// TIA Portal V20 export
FUNCTION_BLOCK "CallEquipment"   // FB8, LAD
TITLE = CallEquipment
AUTHOR : ERsystem_FA2_DH. Kim
// This block contains the logic and futher calls (e.g. sequences, control modules, diagnostics etc.) of the equipment module.
// stored: IsIECCheckEnabled true, MemoryReserve 100, Namespace Unit1.Em0, SetENOAutomatically false
   VAR_INPUT
      ZoneOperationEnable { ExternalWritable := 'False'} : "LWONIK_typeSafetyZoneManualOperation";
   END_VAR
   VAR_IN_OUT
      unitStatus : "LAF_typeUnitStatus";   // Current unit status o be used in this EM
      unitAlarmDB : "LAF_typeAlarms";   // Summarized EM Alarms for the Unit
      emFeedback : "LUC_typeEmFeedback";   // Feedback of the EM to the Unit
   END_VAR
   VAR
      instSequenceUnwinder { S7_SetPoint := 'True'} : "Unit1.Em0.Sequence_1_SepaUnwinderTop";
      instTopHomeJob1 { S7_SetPoint := 'True'} : "LAF_SelectJob";
      instTopUnwindingJob2 { S7_SetPoint := 'True'} : "LAF_SelectJob";
      instTopStopJob3 { S7_SetPoint := 'True'} : "LAF_SelectJob";
      instTopRewidnigJob4 { S7_SetPoint := 'True'} : "LAF_SelectJob";
      instTopRewidnigJob10 { S7_SetPoint := 'True'} : "LAF_SelectJob";
      instCmTopDirectionCheckSensor { S7_SetPoint := 'True'} : "LBC_DigitalSignalCn";
      instCmUnwinderTopRadiusMeasure { ExternalAccessible := 'False'; ExternalVisible := 'False'; ExternalWritable := 'False'} : "LBC_AnalogInputCn";
      instCmRadiusMeasure { S7_SetPoint := 'True'} : "LER_RadiusMeasure";
      instCmUnwinderTopAxisB { S7_SetPoint := 'True'} : "LBC_Axis64Pos_TecPlcCn";
      instInterlockCmUnwinderTopAxisB { S7_SetPoint := 'True'} : "LER_Axis64Pos_InterlockSummary";
      instCmUnwinderAirShaftTopOnOff { ExternalAccessible := 'False'; ExternalVisible := 'False'; ExternalWritable := 'False'; S7_SetPoint := 'True'} : "LBC_TwoWayActuatorCn";
      instCmUnwinderTopEpcControllerInterface { ExternalAccessible := 'False'; ExternalVisible := 'False'; ExternalWritable := 'False'; S7_SetPoint := 'True'} : "LER_EPC_CON600";
      instManageAlarms { ExternalWritable := 'False'} : "LAF_ManageAlarms";
      instEventsPFE : "Unit1.Em0.EventsPFE";
      instLER_BrakeTestUnwinderTopAxisB { S7_SetPoint := 'True'} : "LER_BrakeTest";
      statUnitStatus { ExternalWritable := 'False'} : "LAF_typeUnitStatus";   // Unit Status used in this EM
      statSlmStatus : Struct
         running { ExternalWritable := 'False'} : Bool;
         powerOff { ExternalWritable := 'False'} : Bool;
      END_STRUCT;
      statAllBrakeTest { ExternalWritable := 'False'} : "LER_typeBrakeTestUnitCommands";
      statTonTime { ExternalAccessible := 'False'; ExternalVisible := 'False'; ExternalWritable := 'False'} : Array[0..1999] of TON_TIME;
      statTofTime { ExternalAccessible := 'False'; ExternalVisible := 'False'; ExternalWritable := 'False'} : Array[0..99] of TOF_TIME;
      statPulse { ExternalAccessible := 'False'; ExternalVisible := 'False'; ExternalWritable := 'False'} : Struct
         miscellaneous : Array[0..99] of Bool;
         workingDone : Struct
            mainPnP : Array[0..99] of Bool;
            alignTable : Array[0..99] of Bool;
            ngPnP : Array[0..99] of Bool;
         END_STRUCT;
         axisEnable : Array[0..99] of Bool;
         brakeTest : Array[0..99] of Bool;
      END_STRUCT;
      statEnableManualCmds : Bool;
      statRcEnableCmds : Bool;
      Scan_on { ExternalAccessible := 'False'; ExternalVisible := 'False'; ExternalWritable := 'False'} : Bool;
      "*** Interlock Axis ***" { ExternalAccessible := 'False'; ExternalVisible := 'False'; ExternalWritable := 'False'} : Bool;
      "UnwinderTopAxisB Home" { S7_SetPoint := 'True'} : "Homing.LER_Axis";
      "UnwinderTopAxisB Jog_CW" { S7_SetPoint := 'True'} : "Jog.LER_Axis";
      "UnwinderTopAxisB Jog_CCW" { S7_SetPoint := 'True'} : "Jog.LER_Axis";
      "UnwinderTopAxisB Position" { S7_SetPoint := 'True'} : Array[0..5] of "Position.LER_Axis";
      "*** Interlock Actuator ******" { ExternalAccessible := 'False'; ExternalVisible := 'False'; ExternalWritable := 'False'} : Bool;
      "UnwinderAirShaftTop On" { S7_SetPoint := 'True'} : "Cylinder.LER_Actuator";
      "UnwinderAirShaftTop Off" { S7_SetPoint := 'True'} : "Cylinder.LER_Actuator";
      AXIS1 : "LER_CM_Name";
      Cylinder1 : "LER_CM_Name";
      citi_Ptrig : Array[0..20] of Bool;
      citiTon : Array[0..20] of TON_TIME;
      citi : Time;
      citiTest : Array[0..20] of Bool;
   END_VAR
   VAR_TEMP
      tempIndex : Int;
      tempScInProduction : Bool;   // Mode Production and StateComplete
      tempScNoProduction : Bool;   // Mode Manual and StateComplete
   END_VAR
   VAR CONSTANT
      delayTime : Time := T#3s;
      TRUE : Bool := TRUE;
      FALSE : Bool := FALSE;
      NO_JOB : DInt;   // No job
      MIN_POSITION_NUMBER : SInt;
      INIT_POSITION_NUMBER : SInt := -1;
   END_VAR
   VAR_TEMP   // added for the SCL form of the ladder/FBD networks
      _w1 : Bool;
      _w2 : Bool;
      _w3 : Bool;
      _w4 : Bool;
      _w5 : Bool;
      _w6 : Bool;
      _w7 : Bool;
      _w8 : Bool;
      _w9 : Bool;
   END_VAR
BEGIN

REGION Network 1: BLOCK INFO HEADER
   // (company) / (C) Copyright (year)
   // ---------------------------------------------------------------------------------
   // Title:                             (Title of this block)
   // Comment/Function: (that is implemented in the block)
   // Library/Family:           (that the source is dedicated to)
   // Author:                        (department / person in charge / contact)
   // Target System:          (test system with FW version)
   // Engineering:              TIA Portal (SW version)
   // Restrictions:               (OB types, etc.)
   // Requirements:           (hardware, technological package, etc.)
   // ---------------------------------------------------------------------------------
   // Change log table:
   // Version          | Date             | Signature      | Expert in charge  | Changes applied ------------------------|----------------------|-------------------------|--------------------------------|-----------------------
   // 001.000.000 | yyyy-mm-dd | 0x00000000 | (name of expert) | First released version
END_REGION

REGION Network 2: DESCRIPTION
   // This is a template block provided by the Automation Framework. It can be used to create an own project.
   // The Block Info Header is prepared to put in your own data.
   // Description of the block could be added here and the docu created by Code2Docu.
END_REGION

REGION Network 3: disableFeedbackHomePos
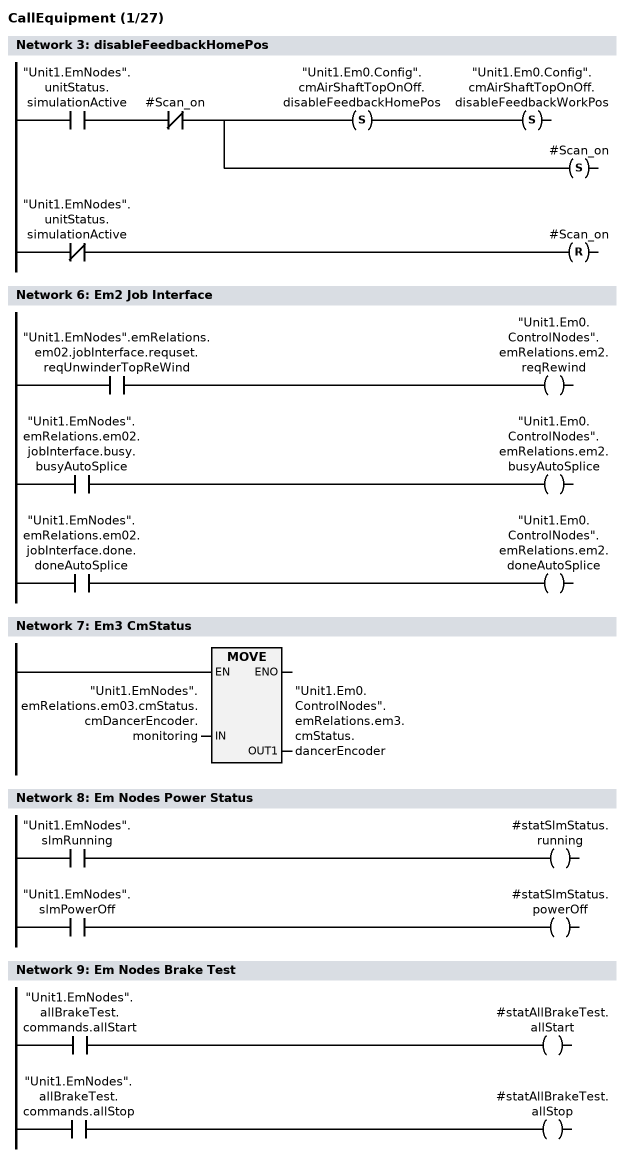
   RUNG wire#powerrail
      Contact( "Unit1.EmNodes".unitStatus.simulationActive )
      I_Contact( #Scan_on )
      wire#w1
      S_Coil( "Unit1.Em0.Config".cmAirShaftTopOnOff.disableFeedbackHomePos )
      S_Coil( "Unit1.Em0.Config".cmAirShaftTopOnOff.disableFeedbackWorkPos )
   END_RUNG
   RUNG wire#w1
      S_Coil( #Scan_on )
   END_RUNG
   RUNG wire#powerrail
      I_Contact( "Unit1.EmNodes".unitStatus.simulationActive )
      R_Coil( #Scan_on )
   END_RUNG
   // the same network as SCL:
   IF "Unit1.EmNodes".unitStatus.simulationActive AND NOT #Scan_on THEN
       "Unit1.Em0.Config".cmAirShaftTopOnOff.disableFeedbackHomePos := TRUE;
       "Unit1.Em0.Config".cmAirShaftTopOnOff.disableFeedbackWorkPos := TRUE;
       #Scan_on := TRUE;
   END_IF;
   IF NOT "Unit1.EmNodes".unitStatus.simulationActive THEN #Scan_on := FALSE; END_IF;
END_REGION

REGION Network 4: ******************** Unit Input ********************
END_REGION

REGION Network 5: Em2 Sequence Interface
END_REGION

REGION Network 6: Em2 Job Interface
   RUNG wire#powerrail
      Contact( "Unit1.EmNodes".emRelations.em02.jobInterface.requset.reqUnwinderTopReWind )
      Coil( "Unit1.Em0.ControlNodes".emRelations.em2.reqRewind )
   END_RUNG
   RUNG wire#powerrail
      Contact( "Unit1.EmNodes".emRelations.em02.jobInterface.busy.busyAutoSplice )
      Coil( "Unit1.Em0.ControlNodes".emRelations.em2.busyAutoSplice )
   END_RUNG
   RUNG wire#powerrail
      Contact( "Unit1.EmNodes".emRelations.em02.jobInterface.done.doneAutoSplice )
      Coil( "Unit1.Em0.ControlNodes".emRelations.em2.doneAutoSplice )
   END_RUNG
   // the same network as SCL:
   "Unit1.Em0.ControlNodes".emRelations.em2.reqRewind := "Unit1.EmNodes".emRelations.em02.jobInterface.requset.reqUnwinderTopReWind;
   "Unit1.Em0.ControlNodes".emRelations.em2.busyAutoSplice := "Unit1.EmNodes".emRelations.em02.jobInterface.busy.busyAutoSplice;
   "Unit1.Em0.ControlNodes".emRelations.em2.doneAutoSplice := "Unit1.EmNodes".emRelations.em02.jobInterface.done.doneAutoSplice;
END_REGION

REGION Network 7: Em3 CmStatus
   RUNG wire#powerrail
      Move(in := "Unit1.EmNodes".emRelations.em03.cmStatus.cmDancerEncoder.monitoring, out1 => "Unit1.Em0.ControlNodes".emRelations.em3.cmStatus.dancerEncoder)
   END_RUNG
   // the same network as SCL:
   "Unit1.Em0.ControlNodes".emRelations.em3.cmStatus.dancerEncoder := "Unit1.EmNodes".emRelations.em03.cmStatus.cmDancerEncoder.monitoring;
END_REGION

REGION Network 8: Em Nodes Power Status
   RUNG wire#powerrail
      Contact( "Unit1.EmNodes".slmRunning )
      Coil( #statSlmStatus.running )
   END_RUNG
   RUNG wire#powerrail
      Contact( "Unit1.EmNodes".slmPowerOff )
      Coil( #statSlmStatus.powerOff )
   END_RUNG
   // the same network as SCL:
   #statSlmStatus.running := "Unit1.EmNodes".slmRunning;
   #statSlmStatus.powerOff := "Unit1.EmNodes".slmPowerOff;
END_REGION

REGION Network 9: Em Nodes Brake Test
   RUNG wire#powerrail
      Contact( "Unit1.EmNodes".allBrakeTest.commands.allStart )
      Coil( #statAllBrakeTest.allStart )
   END_RUNG
   RUNG wire#powerrail
      Contact( "Unit1.EmNodes".allBrakeTest.commands.allStop )
      Coil( #statAllBrakeTest.allStop )
   END_RUNG
   // the same network as SCL:
   #statAllBrakeTest.allStart := "Unit1.EmNodes".allBrakeTest.commands.allStart;
   #statAllBrakeTest.allStop := "Unit1.EmNodes".allBrakeTest.commands.allStop;
END_REGION

REGION Network 10: *************** Equipment Control **************************
END_REGION

REGION Network 11: Interlink EM to Unit
   // This block links and unlinks the EM from the unit. The command to link/unlink can be set directly by the inputs of the block (e.g. to link/unlink based on any program logic) or through the InOut "hmiInterface". The block changes the output "isLinked" to true/false, depending on the command and if a change is allowed. A changed is allowed if the unit is in state aborted, clearing or stopped. The output "isLinked" is send back to the unit. If the EM is not linked, the unit ignores this EM.
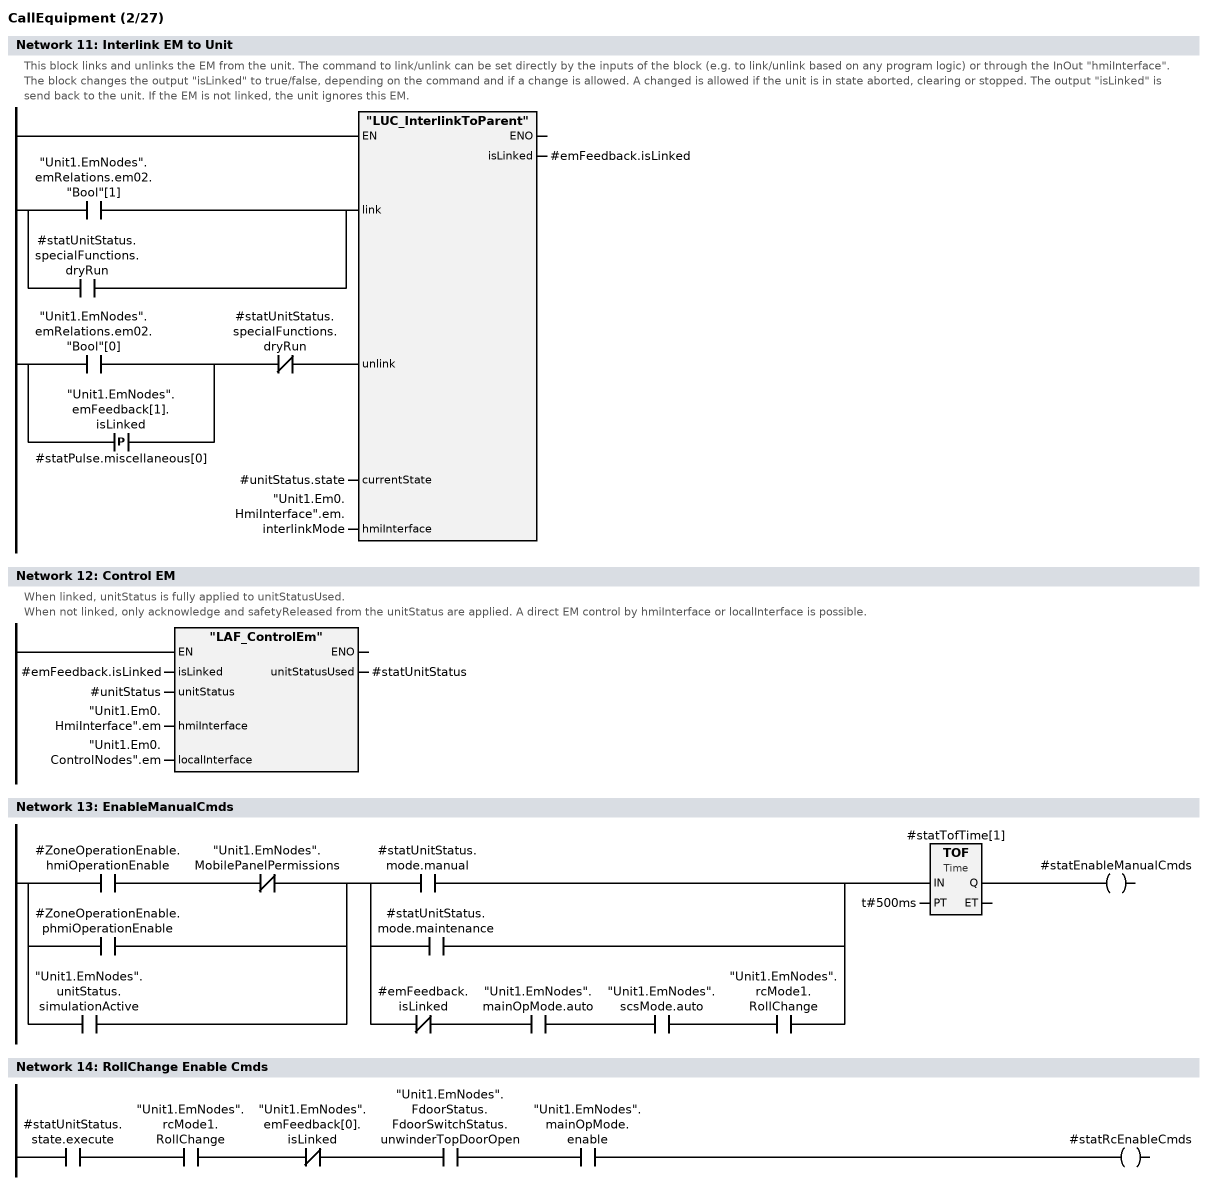
   RUNG wire#powerrail
      "LUC_InterlinkToParent"(link := wire#w1, unlink := wire#w3, currentState := #unitStatus.state, hmiInterface := "Unit1.Em0.HmiInterface".em.interlinkMode, isLinked => #emFeedback.isLinked)
   END_RUNG
   RUNG wire#powerrail
      Contact( "Unit1.EmNodes".emRelations.em02."Bool"[1] )
   END_RUNG wire#w1
   RUNG wire#powerrail
      Contact( #statUnitStatus.specialFunctions.dryRun )
   END_RUNG wire#w1
   RUNG wire#powerrail
      Contact( "Unit1.EmNodes".emRelations.em02."Bool"[0] )
      wire#w2
      I_Contact( #statUnitStatus.specialFunctions.dryRun )
   END_RUNG wire#w3
   RUNG wire#powerrail
      P_Contact(operand := "Unit1.EmNodes".emFeedback[1].isLinked, bit := #statPulse.miscellaneous[0])
   END_RUNG wire#w2
   // the same network as SCL:
   #_w1 := "Unit1.EmNodes".emFeedback[1].isLinked AND NOT #statPulse.miscellaneous[0];   // rising edge of "Unit1.EmNodes".emFeedback[1].isLinked
   #statPulse.miscellaneous[0] := "Unit1.EmNodes".emFeedback[1].isLinked;
   "LUC_InterlinkToParent"(link := "Unit1.EmNodes".emRelations.em02."Bool"[1] OR #statUnitStatus.specialFunctions.dryRun,
                           unlink := ("Unit1.EmNodes".emRelations.em02."Bool"[0] OR #_w1) AND NOT #statUnitStatus.specialFunctions.dryRun,
                           currentState := #unitStatus.state,
                           hmiInterface := "Unit1.Em0.HmiInterface".em.interlinkMode,
                           isLinked => #emFeedback.isLinked);
END_REGION

REGION Network 12: Control EM
   // When linked, unitStatus is fully applied to unitStatusUsed.
   // When not linked, only acknowledge and safetyReleased from the unitStatus are applied. A direct EM control by hmiInterface or localInterface is possible.
   RUNG wire#powerrail
      "LAF_ControlEm"(isLinked := #emFeedback.isLinked, unitStatus := #unitStatus, hmiInterface := "Unit1.Em0.HmiInterface".em, localInterface := "Unit1.Em0.ControlNodes".em, unitStatusUsed => #statUnitStatus)
   END_RUNG
   // the same network as SCL:
   "LAF_ControlEm"(isLinked := #emFeedback.isLinked,
                   unitStatus := #unitStatus,
                   hmiInterface := "Unit1.Em0.HmiInterface".em,
                   localInterface := "Unit1.Em0.ControlNodes".em,
                   unitStatusUsed => #statUnitStatus);
END_REGION

REGION Network 13: EnableManualCmds
   RUNG wire#powerrail
      Contact( #ZoneOperationEnable.hmiOperationEnable )
      I_Contact( "Unit1.EmNodes".MobilePanelPermissions )
      wire#w1
      Contact( #statUnitStatus.mode.manual )
      wire#w2
      { S7_Templates := "time_type := Time" } #statTofTime[1].TOF(pt := t#500ms, et =>)
      Coil( #statEnableManualCmds )
   END_RUNG
   RUNG wire#powerrail
      Contact( #ZoneOperationEnable.phmiOperationEnable )
   END_RUNG wire#w1
   RUNG wire#powerrail
      Contact( "Unit1.EmNodes".unitStatus.simulationActive )
   END_RUNG wire#w1
   RUNG wire#w1
      Contact( #statUnitStatus.mode.maintenance )
   END_RUNG wire#w2
   RUNG wire#w1
      I_Contact( #emFeedback.isLinked )
      Contact( "Unit1.EmNodes".mainOpMode.auto )
      Contact( "Unit1.EmNodes".scsMode.auto )
      Contact( "Unit1.EmNodes".rcMode1.RollChange )
   END_RUNG wire#w2
   // the same network as SCL:
   #statTofTime[1].TOF(IN := ((#ZoneOperationEnable.hmiOperationEnable AND NOT "Unit1.EmNodes".MobilePanelPermissions) OR #ZoneOperationEnable.phmiOperationEnable OR "Unit1.EmNodes".unitStatus.simulationActive) AND (#statUnitStatus.mode.manual OR #statUnitStatus.mode.maintenance OR (NOT #emFeedback.isLinked AND "Unit1.EmNodes".mainOpMode.auto AND "Unit1.EmNodes".scsMode.auto AND "Unit1.EmNodes".rcMode1.RollChange)),
                       PT := t#500ms);
   #statEnableManualCmds := #statTofTime[1].Q;
END_REGION

REGION Network 14: RollChange Enable Cmds
   RUNG wire#powerrail
      Contact( #statUnitStatus.state.execute )
      Contact( "Unit1.EmNodes".rcMode1.RollChange )
      I_Contact( "Unit1.EmNodes".emFeedback[0].isLinked )
      Contact( "Unit1.EmNodes".FdoorStatus.FdoorSwitchStatus.unwinderTopDoorOpen )
      Contact( "Unit1.EmNodes".mainOpMode.enable )
      Coil( #statRcEnableCmds )
   END_RUNG
   // the same network as SCL:
   #statRcEnableCmds := #statUnitStatus.state.execute AND "Unit1.EmNodes".rcMode1.RollChange AND NOT "Unit1.EmNodes".emFeedback[0].isLinked AND "Unit1.EmNodes".FdoorStatus.FdoorSwitchStatus.unwinderTopDoorOpen AND "Unit1.EmNodes".mainOpMode.enable;
END_REGION

REGION Network 15: *************** Control Modules (Sensors) ********************
   // Call control modules that are sensors before the em logic (jobs and sequence), so that the latest value is used in the logic.
END_REGION

REGION Network 16: Call instCmTopDirectionCheckSensor (LBC_DigitalSignal)
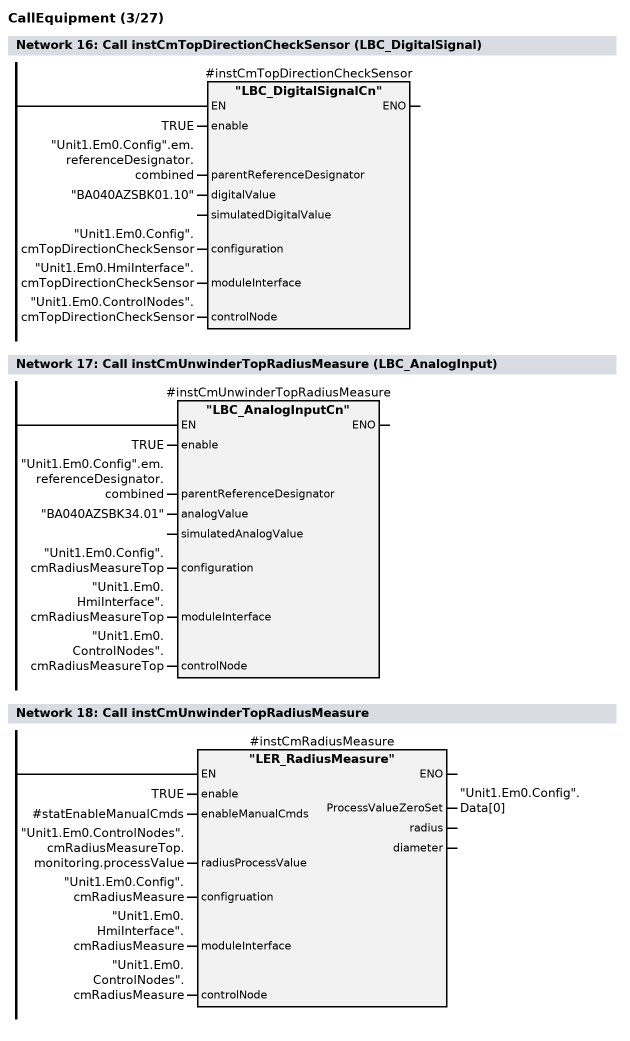
   RUNG wire#powerrail
      #instCmTopDirectionCheckSensor(enable := TRUE, parentReferenceDesignator := "Unit1.Em0.Config".em.referenceDesignator.combined, digitalValue := "BA040AZSBK01.10", simulatedDigitalValue :=, configuration := "Unit1.Em0.Config".cmTopDirectionCheckSensor, moduleInterface := "Unit1.Em0.HmiInterface".cmTopDirectionCheckSensor, controlNode := "Unit1.Em0.ControlNodes".cmTopDirectionCheckSensor)
   END_RUNG
   // the same network as SCL:
   #instCmTopDirectionCheckSensor(enable := TRUE,   // "LBC_DigitalSignalCn"
                           parentReferenceDesignator := "Unit1.Em0.Config".em.referenceDesignator.combined,
                           digitalValue := "BA040AZSBK01.10",
                           configuration := "Unit1.Em0.Config".cmTopDirectionCheckSensor,
                           moduleInterface := "Unit1.Em0.HmiInterface".cmTopDirectionCheckSensor,
                           controlNode := "Unit1.Em0.ControlNodes".cmTopDirectionCheckSensor);
END_REGION

REGION Network 17: Call instCmUnwinderTopRadiusMeasure (LBC_AnalogInput)
   RUNG wire#powerrail
      #instCmUnwinderTopRadiusMeasure(enable := TRUE, parentReferenceDesignator := "Unit1.Em0.Config".em.referenceDesignator.combined, analogValue := "BA040AZSBK34.01", simulatedAnalogValue :=, configuration := "Unit1.Em0.Config".cmRadiusMeasureTop, moduleInterface := "Unit1.Em0.HmiInterface".cmRadiusMeasureTop, controlNode := "Unit1.Em0.ControlNodes".cmRadiusMeasureTop)
   END_RUNG
   // the same network as SCL:
   #instCmUnwinderTopRadiusMeasure(enable := TRUE,   // "LBC_AnalogInputCn"
                           parentReferenceDesignator := "Unit1.Em0.Config".em.referenceDesignator.combined,
                           analogValue := "BA040AZSBK34.01",
                           configuration := "Unit1.Em0.Config".cmRadiusMeasureTop,
                           moduleInterface := "Unit1.Em0.HmiInterface".cmRadiusMeasureTop,
                           controlNode := "Unit1.Em0.ControlNodes".cmRadiusMeasureTop);
END_REGION

REGION Network 18: Call instCmUnwinderTopRadiusMeasure
   RUNG wire#powerrail
      #instCmRadiusMeasure(enable := TRUE, enableManualCmds := #statEnableManualCmds, radiusProcessValue := "Unit1.Em0.ControlNodes".cmRadiusMeasureTop.monitoring.processValue, configruation := "Unit1.Em0.Config".cmRadiusMeasure, moduleInterface := "Unit1.Em0.HmiInterface".cmRadiusMeasure, controlNode := "Unit1.Em0.ControlNodes".cmRadiusMeasure, ProcessValueZeroSet => "Unit1.Em0.Config".Data[0], radius =>, diameter =>)
   END_RUNG
   // the same network as SCL:
   #instCmRadiusMeasure(enable := TRUE,   // "LER_RadiusMeasure"
                        enableManualCmds := #statEnableManualCmds,
                        radiusProcessValue := "Unit1.Em0.ControlNodes".cmRadiusMeasureTop.monitoring.processValue,
                        configruation := "Unit1.Em0.Config".cmRadiusMeasure,
                        moduleInterface := "Unit1.Em0.HmiInterface".cmRadiusMeasure,
                        controlNode := "Unit1.Em0.ControlNodes".cmRadiusMeasure,
                        ProcessValueZeroSet => "Unit1.Em0.Config".Data[0]);
END_REGION

REGION Network 19: *************** Equipment Logic ***************************
END_REGION

REGION Network 20: Map Unit Status to Sequence Status
   // This block maps the unit status to the seuqnce status. Thus, it controls the sequence depending on the unit status. E.g. it sets the sequence to automatic when the unit state is in productions. This blocks work perfectly with the sequences provided in the AF. 
   // This typed block (MapUnitStatusToSequence) could be adjusted to specific application requirements or if other, user-defined sequences are used.
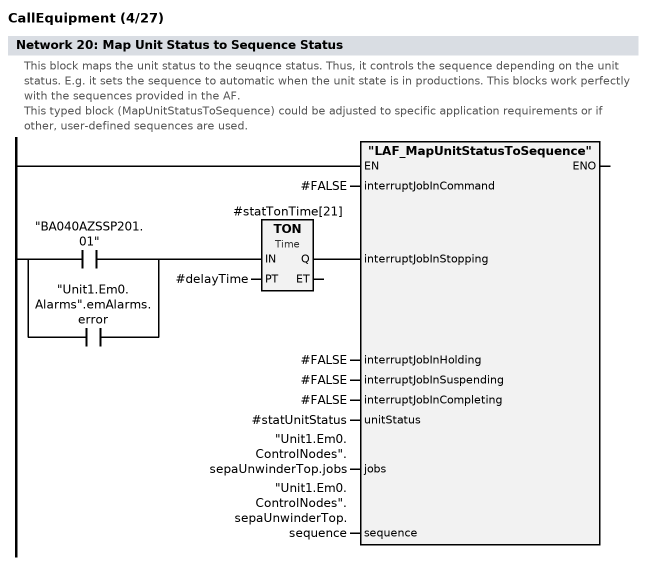
   RUNG wire#powerrail
      "LAF_MapUnitStatusToSequence"(interruptJobInStopping := wire#w2, interruptJobInCommand := #FALSE, interruptJobInHolding := #FALSE, interruptJobInSuspending := #FALSE, interruptJobInCompleting := #FALSE, unitStatus := #statUnitStatus, jobs := "Unit1.Em0.ControlNodes".sepaUnwinderTop.jobs, sequence := "Unit1.Em0.ControlNodes".sepaUnwinderTop.sequence)
   END_RUNG
   RUNG wire#powerrail
      Contact( "BA040AZSSP201.01" )
      wire#w1
      { S7_Templates := "time_type := Time" } #statTonTime[21].TON(pt := #delayTime, et =>)
   END_RUNG wire#w2
   RUNG wire#powerrail
      Contact( "Unit1.Em0.Alarms".emAlarms.error )
   END_RUNG wire#w1
   // the same network as SCL:
   #statTonTime[21].TON(IN := "BA040AZSSP201.01" OR "Unit1.Em0.Alarms".emAlarms.error, PT := #delayTime);
   "LAF_MapUnitStatusToSequence"(interruptJobInCommand := #FALSE,
                           interruptJobInStopping := #statTonTime[21].Q,
                           interruptJobInHolding := #FALSE,
                           interruptJobInSuspending := #FALSE,
                           interruptJobInCompleting := #FALSE,
                           unitStatus := #statUnitStatus,
                           jobs := "Unit1.Em0.ControlNodes".sepaUnwinderTop.jobs,
                           sequence := "Unit1.Em0.ControlNodes".sepaUnwinderTop.sequence);
END_REGION

REGION Network 22: Unwinder Top Select Job
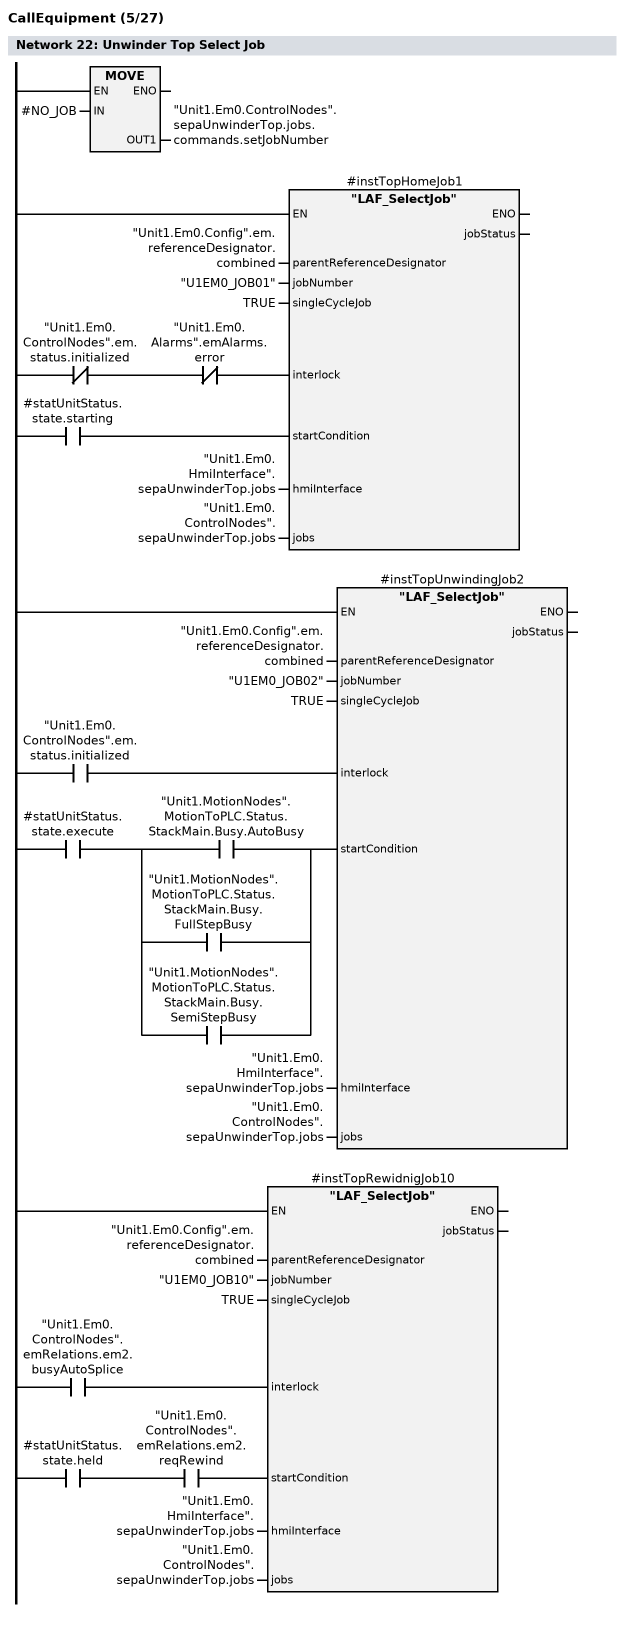
   RUNG wire#powerrail
      Move(in := #NO_JOB, out1 => "Unit1.Em0.ControlNodes".sepaUnwinderTop.jobs.commands.setJobNumber)
   END_RUNG
   RUNG wire#powerrail
      #instTopHomeJob1(interlock := wire#w1, startCondition := wire#w2, parentReferenceDesignator := "Unit1.Em0.Config".em.referenceDesignator.combined, jobNumber := "U1EM0_JOB01", singleCycleJob := TRUE, hmiInterface := "Unit1.Em0.HmiInterface".sepaUnwinderTop.jobs, jobs := "Unit1.Em0.ControlNodes".sepaUnwinderTop.jobs, jobStatus =>)
   END_RUNG
   RUNG wire#powerrail
      I_Contact( "Unit1.Em0.ControlNodes".em.status.initialized )
      I_Contact( "Unit1.Em0.Alarms".emAlarms.error )
   END_RUNG wire#w1
   RUNG wire#powerrail
      Contact( #statUnitStatus.state.starting )
   END_RUNG wire#w2
   RUNG wire#powerrail
      #instTopUnwindingJob2(interlock := wire#w3, startCondition := wire#w5, parentReferenceDesignator := "Unit1.Em0.Config".em.referenceDesignator.combined, jobNumber := "U1EM0_JOB02", singleCycleJob := TRUE, hmiInterface := "Unit1.Em0.HmiInterface".sepaUnwinderTop.jobs, jobs := "Unit1.Em0.ControlNodes".sepaUnwinderTop.jobs, jobStatus =>)
   END_RUNG
   RUNG wire#powerrail
      Contact( "Unit1.Em0.ControlNodes".em.status.initialized )
   END_RUNG wire#w3
   RUNG wire#powerrail
      Contact( #statUnitStatus.state.execute )
      wire#w4
      Contact( "Unit1.MotionNodes".MotionToPLC.Status.StackMain.Busy.AutoBusy )
   END_RUNG wire#w5
   RUNG wire#w4
      Contact( "Unit1.MotionNodes".MotionToPLC.Status.StackMain.Busy.FullStepBusy )
   END_RUNG wire#w5
   RUNG wire#w4
      Contact( "Unit1.MotionNodes".MotionToPLC.Status.StackMain.Busy.SemiStepBusy )
   END_RUNG wire#w5
   RUNG wire#powerrail
      #instTopRewidnigJob10(interlock := wire#w6, startCondition := wire#w7, parentReferenceDesignator := "Unit1.Em0.Config".em.referenceDesignator.combined, jobNumber := "U1EM0_JOB10", singleCycleJob := TRUE, hmiInterface := "Unit1.Em0.HmiInterface".sepaUnwinderTop.jobs, jobs := "Unit1.Em0.ControlNodes".sepaUnwinderTop.jobs, jobStatus =>)
   END_RUNG
   RUNG wire#powerrail
      Contact( "Unit1.Em0.ControlNodes".emRelations.em2.busyAutoSplice )
   END_RUNG wire#w6
   RUNG wire#powerrail
      Contact( #statUnitStatus.state.held )
      Contact( "Unit1.Em0.ControlNodes".emRelations.em2.reqRewind )
   END_RUNG wire#w7
   // the same network as SCL:
   "Unit1.Em0.ControlNodes".sepaUnwinderTop.jobs.commands.setJobNumber := #NO_JOB;
   #instTopHomeJob1(parentReferenceDesignator := "Unit1.Em0.Config".em.referenceDesignator.combined,   // "LAF_SelectJob"
                    jobNumber := "U1EM0_JOB01",
                    singleCycleJob := TRUE,
                    interlock := NOT "Unit1.Em0.ControlNodes".em.status.initialized AND NOT "Unit1.Em0.Alarms".emAlarms.error,
                    startCondition := #statUnitStatus.state.starting,
                    hmiInterface := "Unit1.Em0.HmiInterface".sepaUnwinderTop.jobs,
                    jobs := "Unit1.Em0.ControlNodes".sepaUnwinderTop.jobs);
   #instTopUnwindingJob2(parentReferenceDesignator := "Unit1.Em0.Config".em.referenceDesignator.combined,   // "LAF_SelectJob"
                         jobNumber := "U1EM0_JOB02",
                         singleCycleJob := TRUE,
                         interlock := "Unit1.Em0.ControlNodes".em.status.initialized,
                         startCondition := #statUnitStatus.state.execute AND ("Unit1.MotionNodes".MotionToPLC.Status.StackMain.Busy.AutoBusy OR "Unit1.MotionNodes".MotionToPLC.Status.StackMain.Busy.FullStepBusy OR "Unit1.MotionNodes".MotionToPLC.Status.StackMain.Busy.SemiStepBusy),
                         hmiInterface := "Unit1.Em0.HmiInterface".sepaUnwinderTop.jobs,
                         jobs := "Unit1.Em0.ControlNodes".sepaUnwinderTop.jobs);
   #instTopRewidnigJob10(parentReferenceDesignator := "Unit1.Em0.Config".em.referenceDesignator.combined,   // "LAF_SelectJob"
                         jobNumber := "U1EM0_JOB10",
                         singleCycleJob := TRUE,
                         interlock := "Unit1.Em0.ControlNodes".emRelations.em2.busyAutoSplice,
                         startCondition := #statUnitStatus.state.held AND "Unit1.Em0.ControlNodes".emRelations.em2.reqRewind,
                         hmiInterface := "Unit1.Em0.HmiInterface".sepaUnwinderTop.jobs,
                         jobs := "Unit1.Em0.ControlNodes".sepaUnwinderTop.jobs);
END_REGION

REGION Network 23: Unwinder Top Job Interface [Auto Splicing]
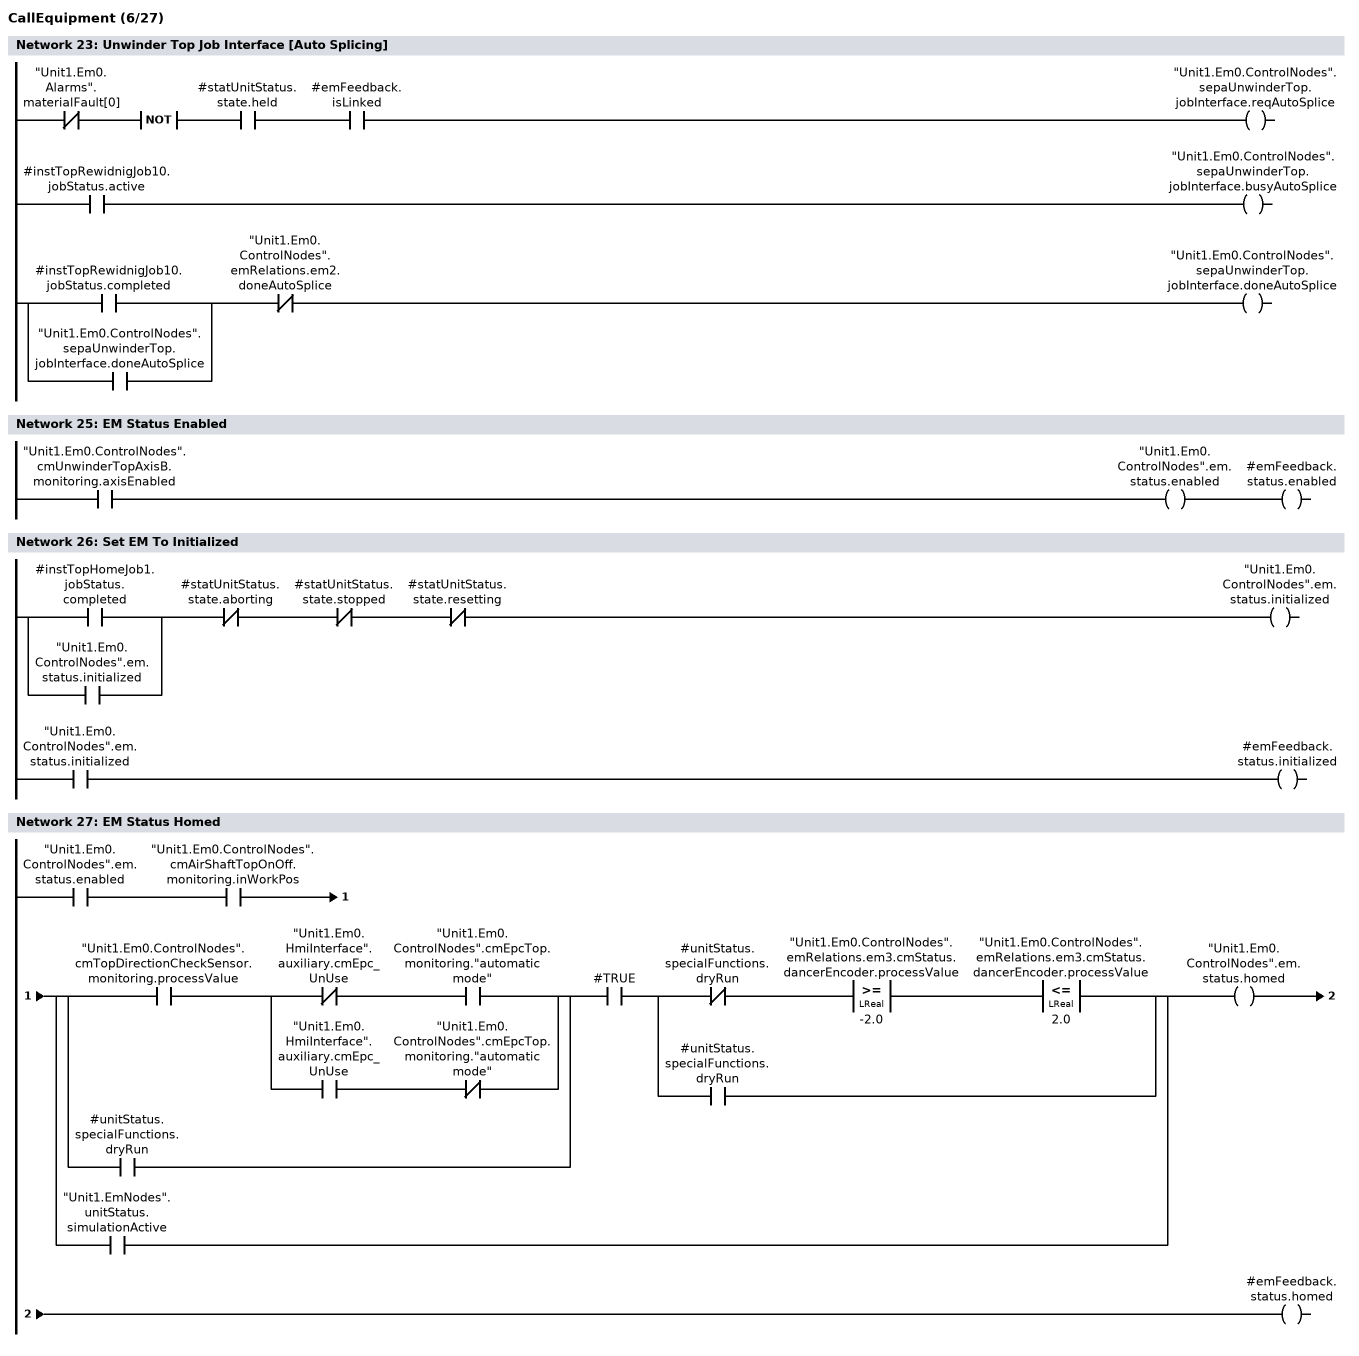
   RUNG wire#powerrail
      I_Contact( "Unit1.Em0.Alarms".materialFault[0] )
      Not()
      Contact( #statUnitStatus.state.held )
      Contact( #emFeedback.isLinked )
      Coil( "Unit1.Em0.ControlNodes".sepaUnwinderTop.jobInterface.reqAutoSplice )
   END_RUNG
   RUNG wire#powerrail
      Contact( #instTopRewidnigJob10.jobStatus.active )
      Coil( "Unit1.Em0.ControlNodes".sepaUnwinderTop.jobInterface.busyAutoSplice )
   END_RUNG
   RUNG wire#powerrail
      Contact( #instTopRewidnigJob10.jobStatus.completed )
      wire#w1
      I_Contact( "Unit1.Em0.ControlNodes".emRelations.em2.doneAutoSplice )
      Coil( "Unit1.Em0.ControlNodes".sepaUnwinderTop.jobInterface.doneAutoSplice )
   END_RUNG
   RUNG wire#powerrail
      Contact( "Unit1.Em0.ControlNodes".sepaUnwinderTop.jobInterface.doneAutoSplice )
   END_RUNG wire#w1
   // the same network as SCL:
   "Unit1.Em0.ControlNodes".sepaUnwinderTop.jobInterface.reqAutoSplice := NOT (NOT "Unit1.Em0.Alarms".materialFault[0]) AND #statUnitStatus.state.held AND #emFeedback.isLinked;
   "Unit1.Em0.ControlNodes".sepaUnwinderTop.jobInterface.busyAutoSplice := #instTopRewidnigJob10.jobStatus.active;
   "Unit1.Em0.ControlNodes".sepaUnwinderTop.jobInterface.doneAutoSplice := (#instTopRewidnigJob10.jobStatus.completed OR "Unit1.Em0.ControlNodes".sepaUnwinderTop.jobInterface.doneAutoSplice) AND NOT "Unit1.Em0.ControlNodes".emRelations.em2.doneAutoSplice;
END_REGION

REGION Network 25: EM Status Enabled
   RUNG wire#powerrail
      Contact( "Unit1.Em0.ControlNodes".cmUnwinderTopAxisB.monitoring.axisEnabled )
      Coil( "Unit1.Em0.ControlNodes".em.status.enabled )
      Coil( #emFeedback.status.enabled )
   END_RUNG
   // the same network as SCL:
   "Unit1.Em0.ControlNodes".em.status.enabled := "Unit1.Em0.ControlNodes".cmUnwinderTopAxisB.monitoring.axisEnabled;
   #emFeedback.status.enabled := "Unit1.Em0.ControlNodes".cmUnwinderTopAxisB.monitoring.axisEnabled;
END_REGION

REGION Network 26: Set EM To Initialized
   RUNG wire#powerrail
      Contact( #instTopHomeJob1.jobStatus.completed )
      wire#w1
      I_Contact( #statUnitStatus.state.aborting )
      I_Contact( #statUnitStatus.state.stopped )
      I_Contact( #statUnitStatus.state.resetting )
      Coil( "Unit1.Em0.ControlNodes".em.status.initialized )
   END_RUNG
   RUNG wire#powerrail
      Contact( "Unit1.Em0.ControlNodes".em.status.initialized )
   END_RUNG wire#w1
   RUNG wire#powerrail
      Contact( "Unit1.Em0.ControlNodes".em.status.initialized )
      Coil( #emFeedback.status.initialized )
   END_RUNG
   // the same network as SCL:
   "Unit1.Em0.ControlNodes".em.status.initialized := (#instTopHomeJob1.jobStatus.completed OR "Unit1.Em0.ControlNodes".em.status.initialized) AND NOT #statUnitStatus.state.aborting AND NOT #statUnitStatus.state.stopped AND NOT #statUnitStatus.state.resetting;
   #emFeedback.status.initialized := "Unit1.Em0.ControlNodes".em.status.initialized;
END_REGION

REGION Network 27: EM Status Homed
   RUNG wire#powerrail
      Contact( "Unit1.Em0.ControlNodes".em.status.enabled )
      Contact( "Unit1.Em0.ControlNodes".cmAirShaftTopOnOff.monitoring.inWorkPos )
      wire#w1
      Contact( "Unit1.Em0.ControlNodes".cmTopDirectionCheckSensor.monitoring.processValue )
      wire#w2
      I_Contact( "Unit1.Em0.HmiInterface".auxiliary.cmEpc_UnUse )
      Contact( "Unit1.Em0.ControlNodes".cmEpcTop.monitoring."automatic mode" )
      wire#w3
      Contact( #TRUE )
      wire#w4
      I_Contact( #unitStatus.specialFunctions.dryRun )
      { S7_Templates := "SrcType := LReal" } GE_Contact(in1 := "Unit1.Em0.ControlNodes".emRelations.em3.cmStatus.dancerEncoder.processValue, in2 := -2.0)
      { S7_Templates := "SrcType := LReal" } LE_Contact(in1 := "Unit1.Em0.ControlNodes".emRelations.em3.cmStatus.dancerEncoder.processValue, in2 := 2.0)
      wire#w5
      Coil( "Unit1.Em0.ControlNodes".em.status.homed )
      Coil( #emFeedback.status.homed )
   END_RUNG
   RUNG wire#w2
      Contact( "Unit1.Em0.HmiInterface".auxiliary.cmEpc_UnUse )
      I_Contact( "Unit1.Em0.ControlNodes".cmEpcTop.monitoring."automatic mode" )
   END_RUNG wire#w3
   RUNG wire#w1
      Contact( #unitStatus.specialFunctions.dryRun )
   END_RUNG wire#w3
   RUNG wire#w4
      Contact( #unitStatus.specialFunctions.dryRun )
   END_RUNG wire#w5
   RUNG wire#w1
      Contact( "Unit1.EmNodes".unitStatus.simulationActive )
   END_RUNG wire#w5
   // the same network as SCL:
   "Unit1.Em0.ControlNodes".em.status.homed := "Unit1.Em0.ControlNodes".em.status.enabled AND "Unit1.Em0.ControlNodes".cmAirShaftTopOnOff.monitoring.inWorkPos AND (((("Unit1.Em0.ControlNodes".cmTopDirectionCheckSensor.monitoring.processValue AND ((NOT "Unit1.Em0.HmiInterface".auxiliary.cmEpc_UnUse AND "Unit1.Em0.ControlNodes".cmEpcTop.monitoring."automatic mode") OR ("Unit1.Em0.HmiInterface".auxiliary.cmEpc_UnUse AND NOT "Unit1.Em0.ControlNodes".cmEpcTop.monitoring."automatic mode"))) OR #unitStatus.specialFunctions.dryRun) AND #TRUE AND ((NOT #unitStatus.specialFunctions.dryRun AND ("Unit1.Em0.ControlNodes".emRelations.em3.cmStatus.dancerEncoder.processValue >= (-2.0)) AND ("Unit1.Em0.ControlNodes".emRelations.em3.cmStatus.dancerEncoder.processValue <= 2.0)) OR #unitStatus.specialFunctions.dryRun)) OR "Unit1.EmNodes".unitStatus.simulationActive);
   #emFeedback.status.homed := "Unit1.Em0.ControlNodes".em.status.homed;
END_REGION

REGION Network 29: Call Sequence [Step]
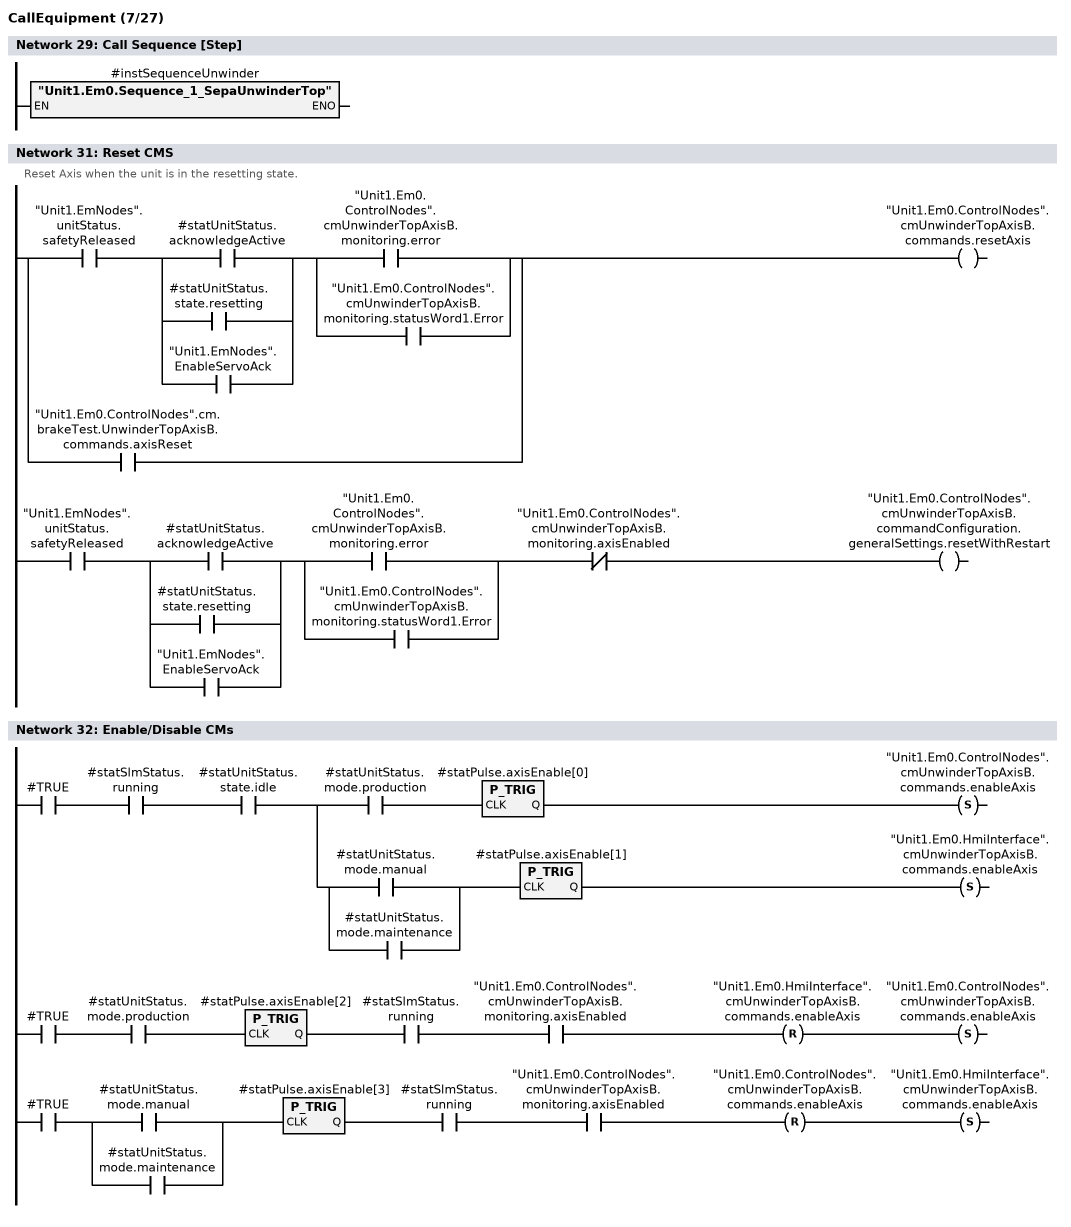
   RUNG wire#powerrail
      #instSequenceUnwinder()
   END_RUNG
   // the same network as SCL:
   #instSequenceUnwinder();   // "Unit1.Em0.Sequence_1_SepaUnwinderTop"
END_REGION

REGION Network 30: ********** Control Modules (Axis) **********
   // Call control modules that are actuators after the em logic (jobs and sequence), so that the latest commands are applied to the actuators.
END_REGION

REGION Network 31: Reset CMS
   // Reset Axis when the unit is in the resetting state.
   RUNG wire#powerrail
      Contact( "Unit1.EmNodes".unitStatus.safetyReleased )
      wire#w1
      Contact( #statUnitStatus.acknowledgeActive )
      wire#w2
      Contact( "Unit1.Em0.ControlNodes".cmUnwinderTopAxisB.monitoring.error )
      wire#w3
      Coil( "Unit1.Em0.ControlNodes".cmUnwinderTopAxisB.commands.resetAxis )
   END_RUNG
   RUNG wire#w1
      Contact( #statUnitStatus.state.resetting )
   END_RUNG wire#w2
   RUNG wire#w1
      Contact( "Unit1.EmNodes".EnableServoAck )
   END_RUNG wire#w2
   RUNG wire#w2
      Contact( "Unit1.Em0.ControlNodes".cmUnwinderTopAxisB.monitoring.statusWord1.Error )
   END_RUNG wire#w3
   RUNG wire#powerrail
      Contact( "Unit1.Em0.ControlNodes".cm.brakeTest.UnwinderTopAxisB.commands.axisReset )
   END_RUNG wire#w3
   RUNG wire#powerrail
      Contact( "Unit1.EmNodes".unitStatus.safetyReleased )
      wire#w4
      Contact( #statUnitStatus.acknowledgeActive )
      wire#w5
      Contact( "Unit1.Em0.ControlNodes".cmUnwinderTopAxisB.monitoring.error )
      wire#w6
      I_Contact( "Unit1.Em0.ControlNodes".cmUnwinderTopAxisB.monitoring.axisEnabled )
      Coil( "Unit1.Em0.ControlNodes".cmUnwinderTopAxisB.commandConfiguration.generalSettings.resetWithRestart )
   END_RUNG
   RUNG wire#w4
      Contact( #statUnitStatus.state.resetting )
   END_RUNG wire#w5
   RUNG wire#w4
      Contact( "Unit1.EmNodes".EnableServoAck )
   END_RUNG wire#w5
   RUNG wire#w5
      Contact( "Unit1.Em0.ControlNodes".cmUnwinderTopAxisB.monitoring.statusWord1.Error )
   END_RUNG wire#w6
   // the same network as SCL:
   "Unit1.Em0.ControlNodes".cmUnwinderTopAxisB.commands.resetAxis := ("Unit1.EmNodes".unitStatus.safetyReleased AND (#statUnitStatus.acknowledgeActive OR #statUnitStatus.state.resetting OR "Unit1.EmNodes".EnableServoAck) AND ("Unit1.Em0.ControlNodes".cmUnwinderTopAxisB.monitoring.error OR "Unit1.Em0.ControlNodes".cmUnwinderTopAxisB.monitoring.statusWord1.Error)) OR "Unit1.Em0.ControlNodes".cm.brakeTest.UnwinderTopAxisB.commands.axisReset;
   "Unit1.Em0.ControlNodes".cmUnwinderTopAxisB.commandConfiguration.generalSettings.resetWithRestart := "Unit1.EmNodes".unitStatus.safetyReleased AND (#statUnitStatus.acknowledgeActive OR #statUnitStatus.state.resetting OR "Unit1.EmNodes".EnableServoAck) AND ("Unit1.Em0.ControlNodes".cmUnwinderTopAxisB.monitoring.error OR "Unit1.Em0.ControlNodes".cmUnwinderTopAxisB.monitoring.statusWord1.Error) AND NOT "Unit1.Em0.ControlNodes".cmUnwinderTopAxisB.monitoring.axisEnabled;
END_REGION

REGION Network 32: Enable/Disable CMs
   RUNG wire#powerrail
      Contact( #TRUE )
      Contact( #statSlmStatus.running )
      Contact( #statUnitStatus.state.idle )
      wire#w1
      Contact( #statUnitStatus.mode.production )
      P_Trig( #statPulse.axisEnable[0] )
      S_Coil( "Unit1.Em0.ControlNodes".cmUnwinderTopAxisB.commands.enableAxis )
   END_RUNG
   RUNG wire#w1
      Contact( #statUnitStatus.mode.manual )
      wire#w2
      P_Trig( #statPulse.axisEnable[1] )
      S_Coil( "Unit1.Em0.HmiInterface".cmUnwinderTopAxisB.commands.enableAxis )
   END_RUNG
   RUNG wire#w1
      Contact( #statUnitStatus.mode.maintenance )
   END_RUNG wire#w2
   RUNG wire#powerrail
      Contact( #TRUE )
      Contact( #statUnitStatus.mode.production )
      P_Trig( #statPulse.axisEnable[2] )
      Contact( #statSlmStatus.running )
      Contact( "Unit1.Em0.ControlNodes".cmUnwinderTopAxisB.monitoring.axisEnabled )
      R_Coil( "Unit1.Em0.HmiInterface".cmUnwinderTopAxisB.commands.enableAxis )
      S_Coil( "Unit1.Em0.ControlNodes".cmUnwinderTopAxisB.commands.enableAxis )
   END_RUNG
   RUNG wire#powerrail
      Contact( #TRUE )
      wire#w3
      Contact( #statUnitStatus.mode.manual )
      wire#w4
      P_Trig( #statPulse.axisEnable[3] )
      Contact( #statSlmStatus.running )
      Contact( "Unit1.Em0.ControlNodes".cmUnwinderTopAxisB.monitoring.axisEnabled )
      R_Coil( "Unit1.Em0.ControlNodes".cmUnwinderTopAxisB.commands.enableAxis )
      S_Coil( "Unit1.Em0.HmiInterface".cmUnwinderTopAxisB.commands.enableAxis )
   END_RUNG
   RUNG wire#w3
      Contact( #statUnitStatus.mode.maintenance )
   END_RUNG wire#w4
   // the same network as SCL:
   #_w1 := #TRUE AND #statSlmStatus.running AND #statUnitStatus.state.idle;
   #_w2 := #_w1 AND #statUnitStatus.mode.production;
   #_w3 := #_w2 AND NOT #statPulse.axisEnable[0];   // rising edge
   #statPulse.axisEnable[0] := #_w2;
   IF #_w3 THEN "Unit1.Em0.ControlNodes".cmUnwinderTopAxisB.commands.enableAxis := TRUE; END_IF;
   #_w4 := #_w1 AND (#statUnitStatus.mode.manual OR #statUnitStatus.mode.maintenance);
   #_w5 := #_w4 AND NOT #statPulse.axisEnable[1];   // rising edge
   #statPulse.axisEnable[1] := #_w4;
   IF #_w5 THEN "Unit1.Em0.HmiInterface".cmUnwinderTopAxisB.commands.enableAxis := TRUE; END_IF;
   #_w6 := #TRUE AND #statUnitStatus.mode.production;
   #_w7 := #_w6 AND NOT #statPulse.axisEnable[2];   // rising edge
   #statPulse.axisEnable[2] := #_w6;
   IF #_w7 AND #statSlmStatus.running AND "Unit1.Em0.ControlNodes".cmUnwinderTopAxisB.monitoring.axisEnabled THEN
       "Unit1.Em0.HmiInterface".cmUnwinderTopAxisB.commands.enableAxis := FALSE;
       "Unit1.Em0.ControlNodes".cmUnwinderTopAxisB.commands.enableAxis := TRUE;
   END_IF;
   #_w8 := #TRUE AND (#statUnitStatus.mode.manual OR #statUnitStatus.mode.maintenance);
   #_w9 := #_w8 AND NOT #statPulse.axisEnable[3];   // rising edge
   #statPulse.axisEnable[3] := #_w8;
   IF #_w9 AND #statSlmStatus.running AND "Unit1.Em0.ControlNodes".cmUnwinderTopAxisB.monitoring.axisEnabled THEN
       "Unit1.Em0.ControlNodes".cmUnwinderTopAxisB.commands.enableAxis := FALSE;
       "Unit1.Em0.HmiInterface".cmUnwinderTopAxisB.commands.enableAxis := TRUE;
   END_IF;
END_REGION

REGION Network 33: PHMI Servo Enable CMs
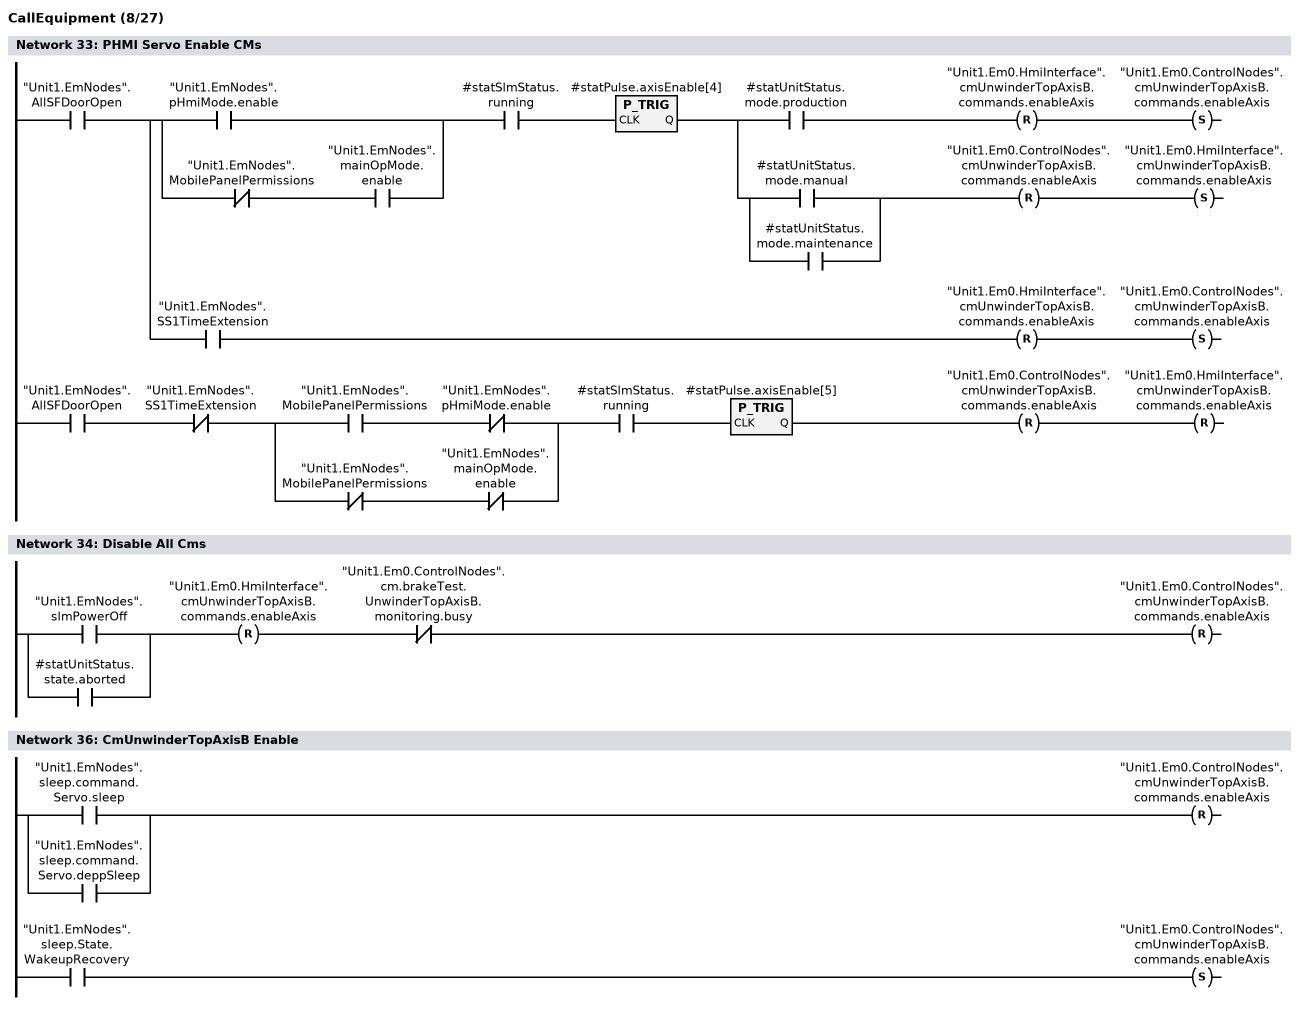
   RUNG wire#powerrail
      Contact( "Unit1.EmNodes".AllSFDoorOpen )
      wire#w1
      Contact( "Unit1.EmNodes".pHmiMode.enable )
      wire#w2
      Contact( #statSlmStatus.running )
      P_Trig( #statPulse.axisEnable[4] )
      wire#w3
      Contact( #statUnitStatus.mode.production )
      R_Coil( "Unit1.Em0.HmiInterface".cmUnwinderTopAxisB.commands.enableAxis )
      S_Coil( "Unit1.Em0.ControlNodes".cmUnwinderTopAxisB.commands.enableAxis )
   END_RUNG
   RUNG wire#w1
      I_Contact( "Unit1.EmNodes".MobilePanelPermissions )
      Contact( "Unit1.EmNodes".mainOpMode.enable )
   END_RUNG wire#w2
   RUNG wire#w3
      Contact( #statUnitStatus.mode.manual )
      wire#w4
      R_Coil( "Unit1.Em0.ControlNodes".cmUnwinderTopAxisB.commands.enableAxis )
      S_Coil( "Unit1.Em0.HmiInterface".cmUnwinderTopAxisB.commands.enableAxis )
   END_RUNG
   RUNG wire#w3
      Contact( #statUnitStatus.mode.maintenance )
   END_RUNG wire#w4
   RUNG wire#w1
      Contact( "Unit1.EmNodes".SS1TimeExtension )
      R_Coil( "Unit1.Em0.HmiInterface".cmUnwinderTopAxisB.commands.enableAxis )
      S_Coil( "Unit1.Em0.ControlNodes".cmUnwinderTopAxisB.commands.enableAxis )
   END_RUNG
   RUNG wire#powerrail
      Contact( "Unit1.EmNodes".AllSFDoorOpen )
      I_Contact( "Unit1.EmNodes".SS1TimeExtension )
      wire#w5
      Contact( "Unit1.EmNodes".MobilePanelPermissions )
      I_Contact( "Unit1.EmNodes".pHmiMode.enable )
      wire#w6
      Contact( #statSlmStatus.running )
      P_Trig( #statPulse.axisEnable[5] )
      R_Coil( "Unit1.Em0.ControlNodes".cmUnwinderTopAxisB.commands.enableAxis )
      R_Coil( "Unit1.Em0.HmiInterface".cmUnwinderTopAxisB.commands.enableAxis )
   END_RUNG
   RUNG wire#w5
      I_Contact( "Unit1.EmNodes".MobilePanelPermissions )
      I_Contact( "Unit1.EmNodes".mainOpMode.enable )
   END_RUNG wire#w6
   // the same network as SCL:
   #_w1 := "Unit1.EmNodes".AllSFDoorOpen AND ("Unit1.EmNodes".pHmiMode.enable OR (NOT "Unit1.EmNodes".MobilePanelPermissions AND "Unit1.EmNodes".mainOpMode.enable)) AND #statSlmStatus.running;
   #_w2 := #_w1 AND NOT #statPulse.axisEnable[4];   // rising edge
   #statPulse.axisEnable[4] := #_w1;
   IF #_w2 AND #statUnitStatus.mode.production THEN
       "Unit1.Em0.HmiInterface".cmUnwinderTopAxisB.commands.enableAxis := FALSE;
       "Unit1.Em0.ControlNodes".cmUnwinderTopAxisB.commands.enableAxis := TRUE;
   END_IF;
   IF #_w2 AND (#statUnitStatus.mode.manual OR #statUnitStatus.mode.maintenance) THEN
       "Unit1.Em0.ControlNodes".cmUnwinderTopAxisB.commands.enableAxis := FALSE;
       "Unit1.Em0.HmiInterface".cmUnwinderTopAxisB.commands.enableAxis := TRUE;
   END_IF;
   IF "Unit1.EmNodes".AllSFDoorOpen AND "Unit1.EmNodes".SS1TimeExtension THEN
       "Unit1.Em0.HmiInterface".cmUnwinderTopAxisB.commands.enableAxis := FALSE;
       "Unit1.Em0.ControlNodes".cmUnwinderTopAxisB.commands.enableAxis := TRUE;
   END_IF;
   #_w3 := "Unit1.EmNodes".AllSFDoorOpen AND NOT "Unit1.EmNodes".SS1TimeExtension AND (("Unit1.EmNodes".MobilePanelPermissions AND NOT "Unit1.EmNodes".pHmiMode.enable) OR (NOT "Unit1.EmNodes".MobilePanelPermissions AND NOT "Unit1.EmNodes".mainOpMode.enable)) AND #statSlmStatus.running;
   #_w4 := #_w3 AND NOT #statPulse.axisEnable[5];   // rising edge
   #statPulse.axisEnable[5] := #_w3;
   IF #_w4 THEN
       "Unit1.Em0.ControlNodes".cmUnwinderTopAxisB.commands.enableAxis := FALSE;
       "Unit1.Em0.HmiInterface".cmUnwinderTopAxisB.commands.enableAxis := FALSE;
   END_IF;
END_REGION

REGION Network 34: Disable All Cms
   RUNG wire#powerrail
      Contact( "Unit1.EmNodes".slmPowerOff )
      wire#w1
      R_Coil( "Unit1.Em0.HmiInterface".cmUnwinderTopAxisB.commands.enableAxis )
      I_Contact( "Unit1.Em0.ControlNodes".cm.brakeTest.UnwinderTopAxisB.monitoring.busy )
      R_Coil( "Unit1.Em0.ControlNodes".cmUnwinderTopAxisB.commands.enableAxis )
   END_RUNG
   RUNG wire#powerrail
      Contact( #statUnitStatus.state.aborted )
   END_RUNG wire#w1
   // the same network as SCL:
   #_w1 := "Unit1.EmNodes".slmPowerOff OR #statUnitStatus.state.aborted;
   IF #_w1 THEN "Unit1.Em0.HmiInterface".cmUnwinderTopAxisB.commands.enableAxis := FALSE; END_IF;
   IF #_w1 AND NOT "Unit1.Em0.ControlNodes".cm.brakeTest.UnwinderTopAxisB.monitoring.busy THEN
       "Unit1.Em0.ControlNodes".cmUnwinderTopAxisB.commands.enableAxis := FALSE;
   END_IF;
END_REGION

REGION Network 36: CmUnwinderTopAxisB Enable
   RUNG wire#powerrail
      Contact( "Unit1.EmNodes".sleep.command.Servo.sleep )
      wire#w1
      R_Coil( "Unit1.Em0.ControlNodes".cmUnwinderTopAxisB.commands.enableAxis )
   END_RUNG
   RUNG wire#powerrail
      Contact( "Unit1.EmNodes".sleep.command.Servo.deppSleep )
   END_RUNG wire#w1
   RUNG wire#powerrail
      Contact( "Unit1.EmNodes".sleep.State.WakeupRecovery )
      S_Coil( "Unit1.Em0.ControlNodes".cmUnwinderTopAxisB.commands.enableAxis )
   END_RUNG
   // the same network as SCL:
   IF "Unit1.EmNodes".sleep.command.Servo.sleep OR "Unit1.EmNodes".sleep.command.Servo.deppSleep THEN
       "Unit1.Em0.ControlNodes".cmUnwinderTopAxisB.commands.enableAxis := FALSE;
   END_IF;
   IF "Unit1.EmNodes".sleep.State.WakeupRecovery THEN
       "Unit1.Em0.ControlNodes".cmUnwinderTopAxisB.commands.enableAxis := TRUE;
   END_IF;
END_REGION

REGION Network 37: Interlock/Servo
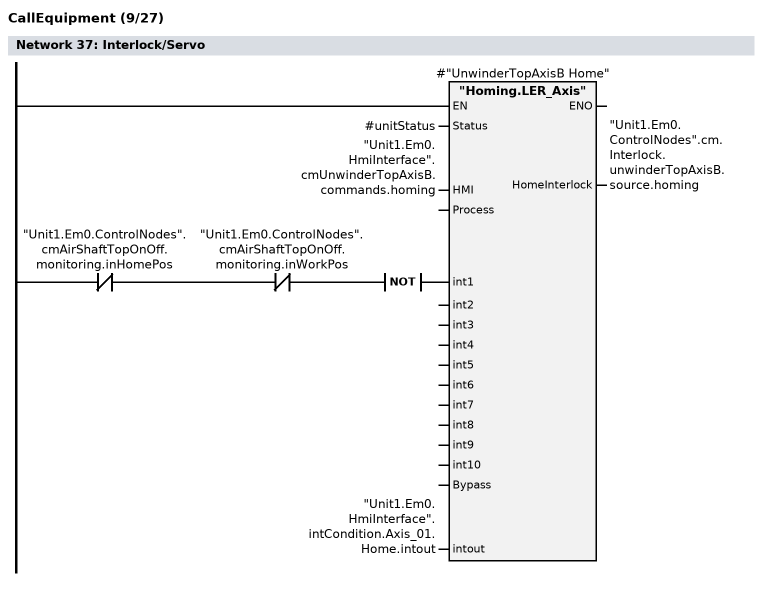
   RUNG wire#powerrail
      #"UnwinderTopAxisB Home"(int1 := wire#w1, Status := #unitStatus, HMI := "Unit1.Em0.HmiInterface".cmUnwinderTopAxisB.commands.homing, Process :=, int2 :=, int3 :=, int4 :=, int5 :=, int6 :=, int7 :=, int8 :=, int9 :=, int10 :=, Bypass :=, intout := "Unit1.Em0.HmiInterface".intCondition.Axis_01.Home.intout, HomeInterlock => "Unit1.Em0.ControlNodes".cm.Interlock.unwinderTopAxisB.source.homing)
   END_RUNG
   RUNG wire#powerrail
      I_Contact( "Unit1.Em0.ControlNodes".cmAirShaftTopOnOff.monitoring.inHomePos )
      I_Contact( "Unit1.Em0.ControlNodes".cmAirShaftTopOnOff.monitoring.inWorkPos )
      Not()
   END_RUNG wire#w1
   // the same network as SCL:
   #"UnwinderTopAxisB Home"(Status := #unitStatus,   // "Homing.LER_Axis"
                           HMI := "Unit1.Em0.HmiInterface".cmUnwinderTopAxisB.commands.homing,
                           int1 := NOT (NOT "Unit1.Em0.ControlNodes".cmAirShaftTopOnOff.monitoring.inHomePos AND NOT "Unit1.Em0.ControlNodes".cmAirShaftTopOnOff.monitoring.inWorkPos),
                           intout := "Unit1.Em0.HmiInterface".intCondition.Axis_01.Home.intout,
                           HomeInterlock => "Unit1.Em0.ControlNodes".cm.Interlock.unwinderTopAxisB.source.homing);
END_REGION

REGION Network 38: CmUnwinderTopAxisB Position Absolute Jog
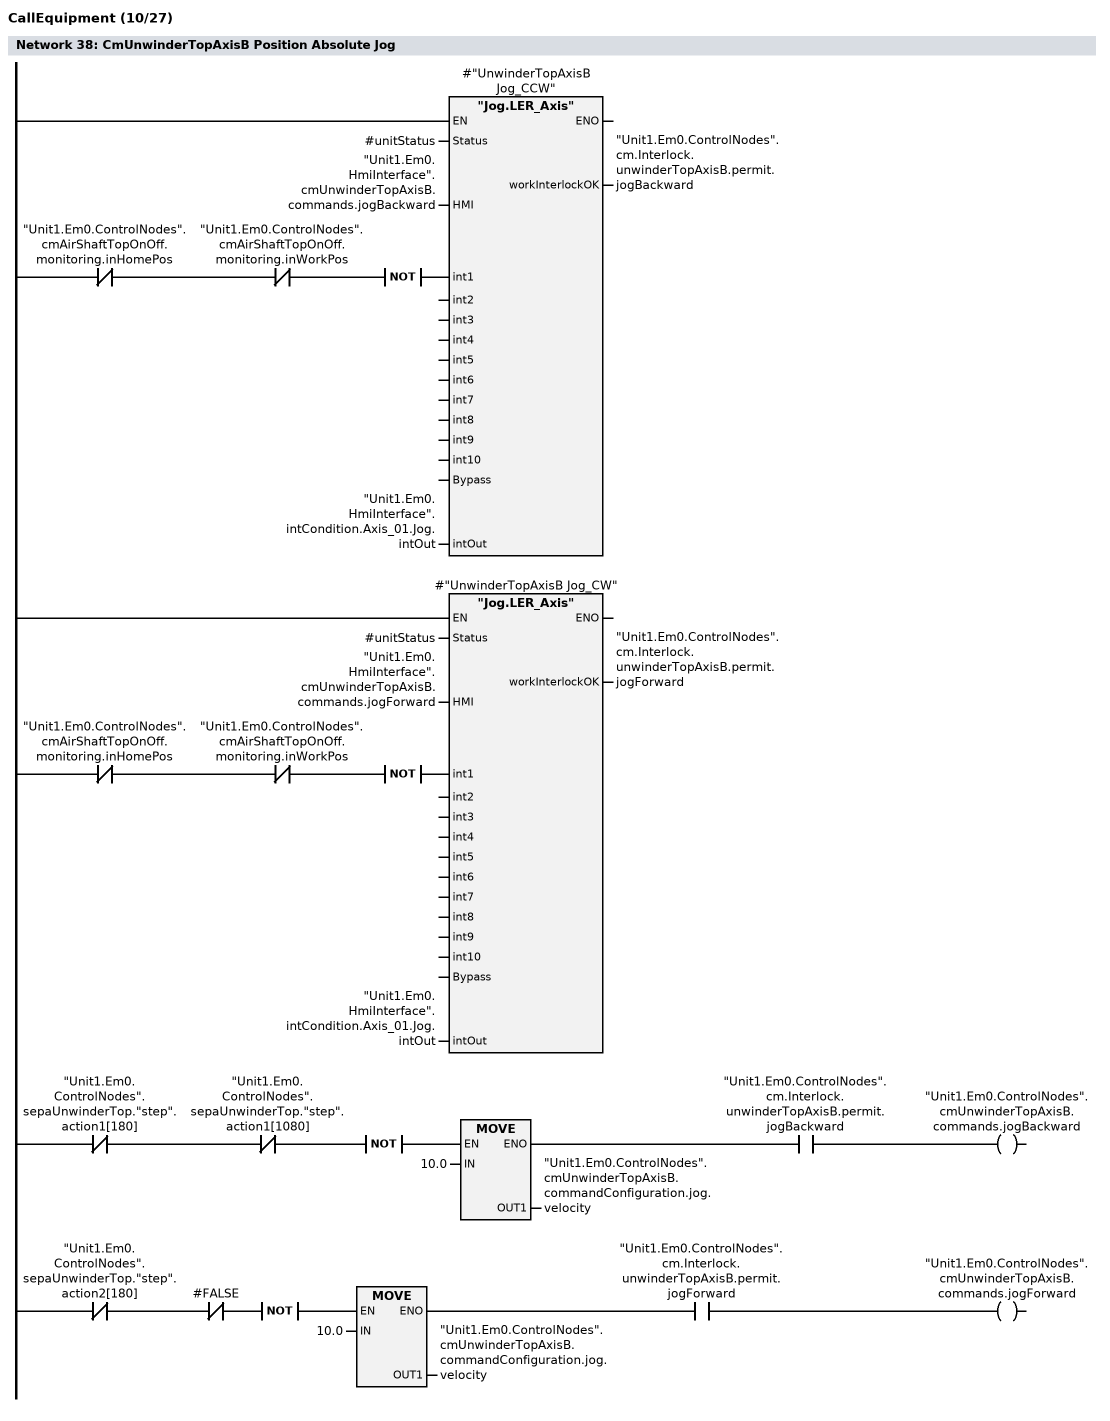
   RUNG wire#powerrail
      #"UnwinderTopAxisB Jog_CCW"(int1 := wire#w1, Status := #unitStatus, HMI := "Unit1.Em0.HmiInterface".cmUnwinderTopAxisB.commands.jogBackward, int2 :=, int3 :=, int4 :=, int5 :=, int6 :=, int7 :=, int8 :=, int9 :=, int10 :=, Bypass :=, intOut := "Unit1.Em0.HmiInterface".intCondition.Axis_01.Jog.intOut, workInterlockOK => "Unit1.Em0.ControlNodes".cm.Interlock.unwinderTopAxisB.permit.jogBackward)
   END_RUNG
   RUNG wire#powerrail
      I_Contact( "Unit1.Em0.ControlNodes".cmAirShaftTopOnOff.monitoring.inHomePos )
      I_Contact( "Unit1.Em0.ControlNodes".cmAirShaftTopOnOff.monitoring.inWorkPos )
      Not()
   END_RUNG wire#w1
   RUNG wire#powerrail
      #"UnwinderTopAxisB Jog_CW"(int1 := wire#w2, Status := #unitStatus, HMI := "Unit1.Em0.HmiInterface".cmUnwinderTopAxisB.commands.jogForward, int2 :=, int3 :=, int4 :=, int5 :=, int6 :=, int7 :=, int8 :=, int9 :=, int10 :=, Bypass :=, intOut := "Unit1.Em0.HmiInterface".intCondition.Axis_01.Jog.intOut, workInterlockOK => "Unit1.Em0.ControlNodes".cm.Interlock.unwinderTopAxisB.permit.jogForward)
   END_RUNG
   RUNG wire#powerrail
      I_Contact( "Unit1.Em0.ControlNodes".cmAirShaftTopOnOff.monitoring.inHomePos )
      I_Contact( "Unit1.Em0.ControlNodes".cmAirShaftTopOnOff.monitoring.inWorkPos )
      Not()
   END_RUNG wire#w2
   RUNG wire#powerrail
      I_Contact( "Unit1.Em0.ControlNodes".sepaUnwinderTop."step".action1[180] )
      I_Contact( "Unit1.Em0.ControlNodes".sepaUnwinderTop."step".action1[1080] )
      Not()
      Move(in := 10.0, out1 => "Unit1.Em0.ControlNodes".cmUnwinderTopAxisB.commandConfiguration.jog.velocity)
      Contact( "Unit1.Em0.ControlNodes".cm.Interlock.unwinderTopAxisB.permit.jogBackward )
      Coil( "Unit1.Em0.ControlNodes".cmUnwinderTopAxisB.commands.jogBackward )
   END_RUNG
   RUNG wire#powerrail
      I_Contact( "Unit1.Em0.ControlNodes".sepaUnwinderTop."step".action2[180] )
      I_Contact( #FALSE )
      Not()
      Move(in := 10.0, out1 => "Unit1.Em0.ControlNodes".cmUnwinderTopAxisB.commandConfiguration.jog.velocity)
      Contact( "Unit1.Em0.ControlNodes".cm.Interlock.unwinderTopAxisB.permit.jogForward )
      Coil( "Unit1.Em0.ControlNodes".cmUnwinderTopAxisB.commands.jogForward )
   END_RUNG
   // the same network as SCL:
   #"UnwinderTopAxisB Jog_CCW"(Status := #unitStatus,   // "Jog.LER_Axis"
                           HMI := "Unit1.Em0.HmiInterface".cmUnwinderTopAxisB.commands.jogBackward,
                           int1 := NOT (NOT "Unit1.Em0.ControlNodes".cmAirShaftTopOnOff.monitoring.inHomePos AND NOT "Unit1.Em0.ControlNodes".cmAirShaftTopOnOff.monitoring.inWorkPos),
                           intOut := "Unit1.Em0.HmiInterface".intCondition.Axis_01.Jog.intOut,
                           workInterlockOK => "Unit1.Em0.ControlNodes".cm.Interlock.unwinderTopAxisB.permit.jogBackward);
   #"UnwinderTopAxisB Jog_CW"(Status := #unitStatus,   // "Jog.LER_Axis"
                           HMI := "Unit1.Em0.HmiInterface".cmUnwinderTopAxisB.commands.jogForward,
                           int1 := NOT (NOT "Unit1.Em0.ControlNodes".cmAirShaftTopOnOff.monitoring.inHomePos AND NOT "Unit1.Em0.ControlNodes".cmAirShaftTopOnOff.monitoring.inWorkPos),
                           intOut := "Unit1.Em0.HmiInterface".intCondition.Axis_01.Jog.intOut,
                           workInterlockOK => "Unit1.Em0.ControlNodes".cm.Interlock.unwinderTopAxisB.permit.jogForward);
   #_w1 := NOT (NOT "Unit1.Em0.ControlNodes".sepaUnwinderTop."step".action1[180] AND NOT "Unit1.Em0.ControlNodes".sepaUnwinderTop."step".action1[1080]);
   IF #_w1 THEN
       "Unit1.Em0.ControlNodes".cmUnwinderTopAxisB.commandConfiguration.jog.velocity := 10.0;
   END_IF;
   "Unit1.Em0.ControlNodes".cmUnwinderTopAxisB.commands.jogBackward := #_w1 AND "Unit1.Em0.ControlNodes".cm.Interlock.unwinderTopAxisB.permit.jogBackward;
   #_w2 := NOT (NOT "Unit1.Em0.ControlNodes".sepaUnwinderTop."step".action2[180] AND NOT #FALSE);
   IF #_w2 THEN
       "Unit1.Em0.ControlNodes".cmUnwinderTopAxisB.commandConfiguration.jog.velocity := 10.0;
   END_IF;
   "Unit1.Em0.ControlNodes".cmUnwinderTopAxisB.commands.jogForward := #_w2 AND "Unit1.Em0.ControlNodes".cm.Interlock.unwinderTopAxisB.permit.jogForward;
END_REGION

REGION Network 39: CmUnwinderTopAxisB Position Absolute Position0
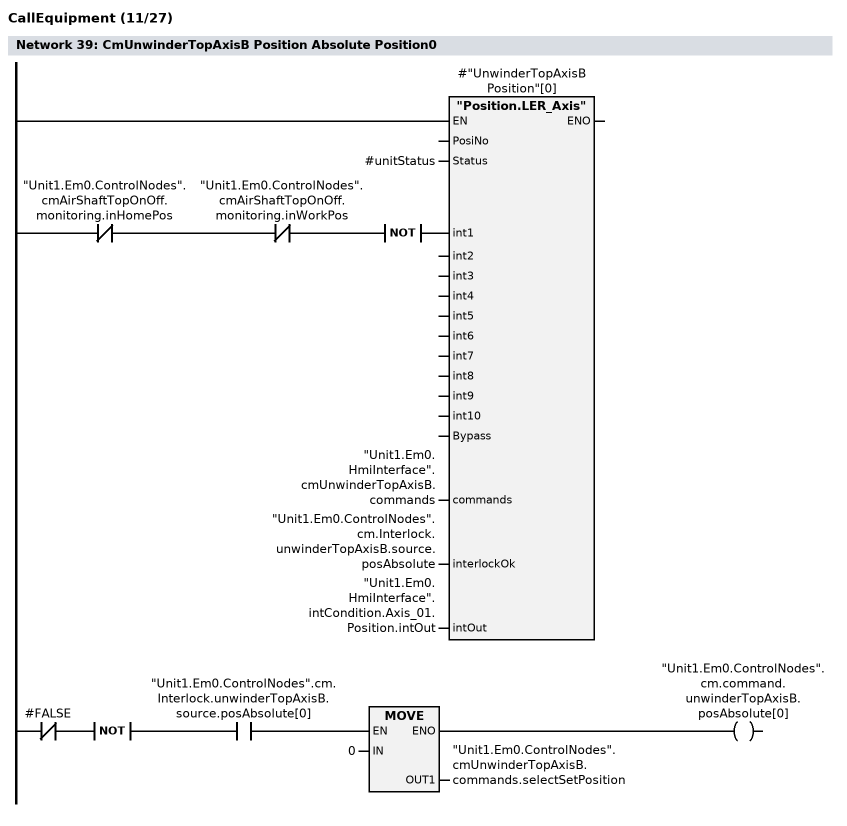
   RUNG wire#powerrail
      #"UnwinderTopAxisB Position"[0](int1 := wire#w1, PosiNo :=, Status := #unitStatus, int2 :=, int3 :=, int4 :=, int5 :=, int6 :=, int7 :=, int8 :=, int9 :=, int10 :=, Bypass :=, commands := "Unit1.Em0.HmiInterface".cmUnwinderTopAxisB.commands, interlockOk := "Unit1.Em0.ControlNodes".cm.Interlock.unwinderTopAxisB.source.posAbsolute, intOut := "Unit1.Em0.HmiInterface".intCondition.Axis_01.Position.intOut)
   END_RUNG
   RUNG wire#powerrail
      I_Contact( "Unit1.Em0.ControlNodes".cmAirShaftTopOnOff.monitoring.inHomePos )
      I_Contact( "Unit1.Em0.ControlNodes".cmAirShaftTopOnOff.monitoring.inWorkPos )
      Not()
   END_RUNG wire#w1
   RUNG wire#powerrail
      I_Contact( #FALSE )
      Not()
      Contact( "Unit1.Em0.ControlNodes".cm.Interlock.unwinderTopAxisB.source.posAbsolute[0] )
      Move(in := 0, out1 => "Unit1.Em0.ControlNodes".cmUnwinderTopAxisB.commands.selectSetPosition)
      Coil( "Unit1.Em0.ControlNodes".cm.command.unwinderTopAxisB.posAbsolute[0] )
   END_RUNG
   // the same network as SCL:
   #"UnwinderTopAxisB Position"[0](Status := #unitStatus,   // "Position.LER_Axis"
                           int1 := NOT (NOT "Unit1.Em0.ControlNodes".cmAirShaftTopOnOff.monitoring.inHomePos AND NOT "Unit1.Em0.ControlNodes".cmAirShaftTopOnOff.monitoring.inWorkPos),
                           commands := "Unit1.Em0.HmiInterface".cmUnwinderTopAxisB.commands,
                           interlockOk := "Unit1.Em0.ControlNodes".cm.Interlock.unwinderTopAxisB.source.posAbsolute,
                           intOut := "Unit1.Em0.HmiInterface".intCondition.Axis_01.Position.intOut);
   #_w1 := NOT (NOT #FALSE) AND "Unit1.Em0.ControlNodes".cm.Interlock.unwinderTopAxisB.source.posAbsolute[0];
   IF #_w1 THEN "Unit1.Em0.ControlNodes".cmUnwinderTopAxisB.commands.selectSetPosition := 0; END_IF;
   "Unit1.Em0.ControlNodes".cm.command.unwinderTopAxisB.posAbsolute[0] := #_w1;
END_REGION

REGION Network 40: CmUnwinderTopAxisB Position Absolute Position1
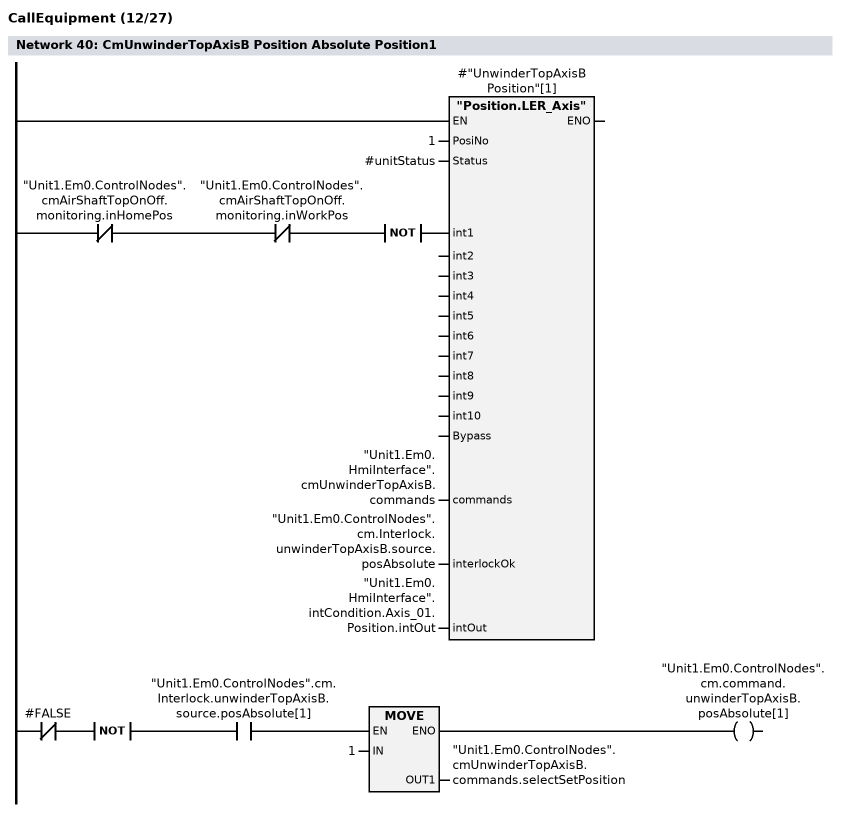
   RUNG wire#powerrail
      #"UnwinderTopAxisB Position"[1](int1 := wire#w1, PosiNo := 1, Status := #unitStatus, int2 :=, int3 :=, int4 :=, int5 :=, int6 :=, int7 :=, int8 :=, int9 :=, int10 :=, Bypass :=, commands := "Unit1.Em0.HmiInterface".cmUnwinderTopAxisB.commands, interlockOk := "Unit1.Em0.ControlNodes".cm.Interlock.unwinderTopAxisB.source.posAbsolute, intOut := "Unit1.Em0.HmiInterface".intCondition.Axis_01.Position.intOut)
   END_RUNG
   RUNG wire#powerrail
      I_Contact( "Unit1.Em0.ControlNodes".cmAirShaftTopOnOff.monitoring.inHomePos )
      I_Contact( "Unit1.Em0.ControlNodes".cmAirShaftTopOnOff.monitoring.inWorkPos )
      Not()
   END_RUNG wire#w1
   RUNG wire#powerrail
      I_Contact( #FALSE )
      Not()
      Contact( "Unit1.Em0.ControlNodes".cm.Interlock.unwinderTopAxisB.source.posAbsolute[1] )
      Move(in := 1, out1 => "Unit1.Em0.ControlNodes".cmUnwinderTopAxisB.commands.selectSetPosition)
      Coil( "Unit1.Em0.ControlNodes".cm.command.unwinderTopAxisB.posAbsolute[1] )
   END_RUNG
   // the same network as SCL:
   #"UnwinderTopAxisB Position"[1](PosiNo := 1,   // "Position.LER_Axis"
                           Status := #unitStatus,
                           int1 := NOT (NOT "Unit1.Em0.ControlNodes".cmAirShaftTopOnOff.monitoring.inHomePos AND NOT "Unit1.Em0.ControlNodes".cmAirShaftTopOnOff.monitoring.inWorkPos),
                           commands := "Unit1.Em0.HmiInterface".cmUnwinderTopAxisB.commands,
                           interlockOk := "Unit1.Em0.ControlNodes".cm.Interlock.unwinderTopAxisB.source.posAbsolute,
                           intOut := "Unit1.Em0.HmiInterface".intCondition.Axis_01.Position.intOut);
   #_w1 := NOT (NOT #FALSE) AND "Unit1.Em0.ControlNodes".cm.Interlock.unwinderTopAxisB.source.posAbsolute[1];
   IF #_w1 THEN "Unit1.Em0.ControlNodes".cmUnwinderTopAxisB.commands.selectSetPosition := 1; END_IF;
   "Unit1.Em0.ControlNodes".cm.command.unwinderTopAxisB.posAbsolute[1] := #_w1;
END_REGION

REGION Network 41: CmUnwinderTopAxisB Position Absolute Position2
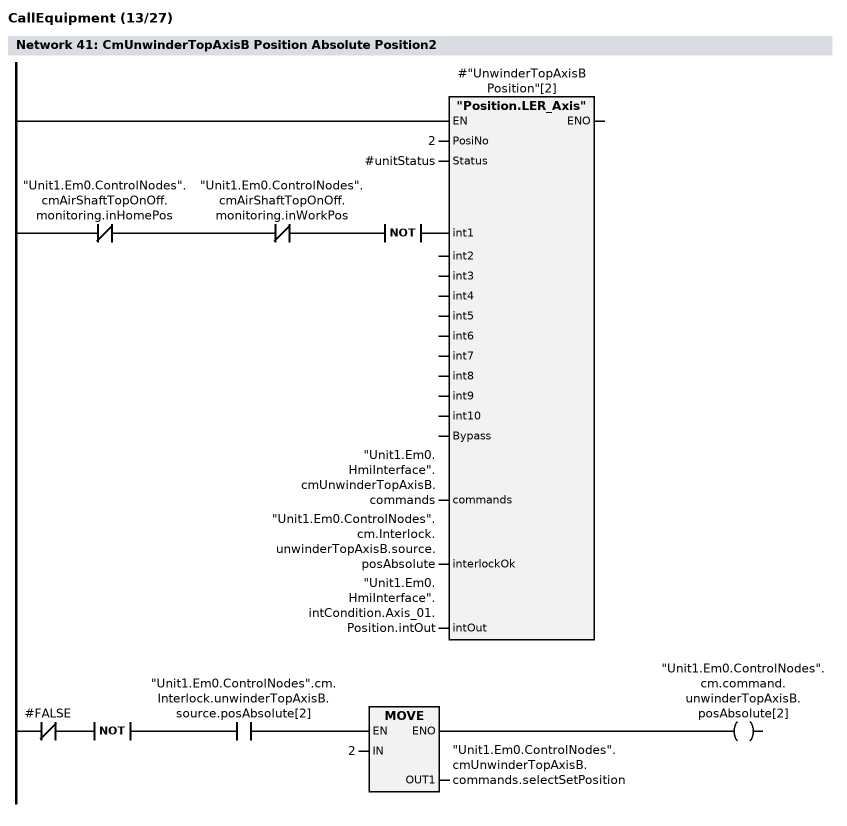
   RUNG wire#powerrail
      #"UnwinderTopAxisB Position"[2](int1 := wire#w1, PosiNo := 2, Status := #unitStatus, int2 :=, int3 :=, int4 :=, int5 :=, int6 :=, int7 :=, int8 :=, int9 :=, int10 :=, Bypass :=, commands := "Unit1.Em0.HmiInterface".cmUnwinderTopAxisB.commands, interlockOk := "Unit1.Em0.ControlNodes".cm.Interlock.unwinderTopAxisB.source.posAbsolute, intOut := "Unit1.Em0.HmiInterface".intCondition.Axis_01.Position.intOut)
   END_RUNG
   RUNG wire#powerrail
      I_Contact( "Unit1.Em0.ControlNodes".cmAirShaftTopOnOff.monitoring.inHomePos )
      I_Contact( "Unit1.Em0.ControlNodes".cmAirShaftTopOnOff.monitoring.inWorkPos )
      Not()
   END_RUNG wire#w1
   RUNG wire#powerrail
      I_Contact( #FALSE )
      Not()
      Contact( "Unit1.Em0.ControlNodes".cm.Interlock.unwinderTopAxisB.source.posAbsolute[2] )
      Move(in := 2, out1 => "Unit1.Em0.ControlNodes".cmUnwinderTopAxisB.commands.selectSetPosition)
      Coil( "Unit1.Em0.ControlNodes".cm.command.unwinderTopAxisB.posAbsolute[2] )
   END_RUNG
   // the same network as SCL:
   #"UnwinderTopAxisB Position"[2](PosiNo := 2,   // "Position.LER_Axis"
                           Status := #unitStatus,
                           int1 := NOT (NOT "Unit1.Em0.ControlNodes".cmAirShaftTopOnOff.monitoring.inHomePos AND NOT "Unit1.Em0.ControlNodes".cmAirShaftTopOnOff.monitoring.inWorkPos),
                           commands := "Unit1.Em0.HmiInterface".cmUnwinderTopAxisB.commands,
                           interlockOk := "Unit1.Em0.ControlNodes".cm.Interlock.unwinderTopAxisB.source.posAbsolute,
                           intOut := "Unit1.Em0.HmiInterface".intCondition.Axis_01.Position.intOut);
   #_w1 := NOT (NOT #FALSE) AND "Unit1.Em0.ControlNodes".cm.Interlock.unwinderTopAxisB.source.posAbsolute[2];
   IF #_w1 THEN "Unit1.Em0.ControlNodes".cmUnwinderTopAxisB.commands.selectSetPosition := 2; END_IF;
   "Unit1.Em0.ControlNodes".cm.command.unwinderTopAxisB.posAbsolute[2] := #_w1;
END_REGION

REGION Network 42: CmUnwinderTopAxisB Position Absolute Position3
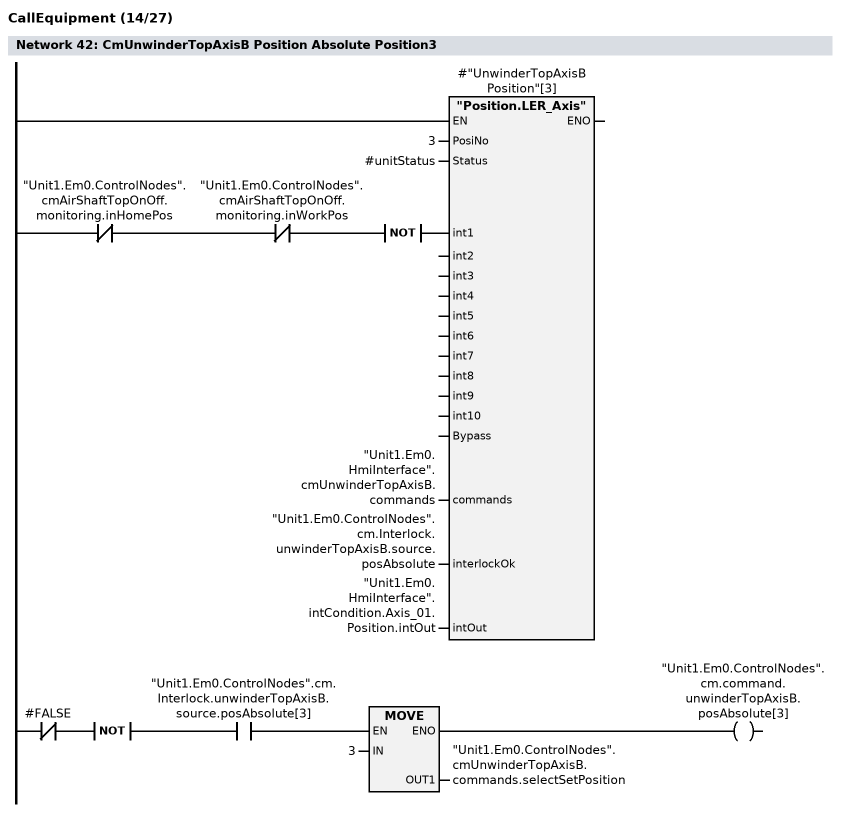
   RUNG wire#powerrail
      #"UnwinderTopAxisB Position"[3](int1 := wire#w1, PosiNo := 3, Status := #unitStatus, int2 :=, int3 :=, int4 :=, int5 :=, int6 :=, int7 :=, int8 :=, int9 :=, int10 :=, Bypass :=, commands := "Unit1.Em0.HmiInterface".cmUnwinderTopAxisB.commands, interlockOk := "Unit1.Em0.ControlNodes".cm.Interlock.unwinderTopAxisB.source.posAbsolute, intOut := "Unit1.Em0.HmiInterface".intCondition.Axis_01.Position.intOut)
   END_RUNG
   RUNG wire#powerrail
      I_Contact( "Unit1.Em0.ControlNodes".cmAirShaftTopOnOff.monitoring.inHomePos )
      I_Contact( "Unit1.Em0.ControlNodes".cmAirShaftTopOnOff.monitoring.inWorkPos )
      Not()
   END_RUNG wire#w1
   RUNG wire#powerrail
      I_Contact( #FALSE )
      Not()
      Contact( "Unit1.Em0.ControlNodes".cm.Interlock.unwinderTopAxisB.source.posAbsolute[3] )
      Move(in := 3, out1 => "Unit1.Em0.ControlNodes".cmUnwinderTopAxisB.commands.selectSetPosition)
      Coil( "Unit1.Em0.ControlNodes".cm.command.unwinderTopAxisB.posAbsolute[3] )
   END_RUNG
   // the same network as SCL:
   #"UnwinderTopAxisB Position"[3](PosiNo := 3,   // "Position.LER_Axis"
                           Status := #unitStatus,
                           int1 := NOT (NOT "Unit1.Em0.ControlNodes".cmAirShaftTopOnOff.monitoring.inHomePos AND NOT "Unit1.Em0.ControlNodes".cmAirShaftTopOnOff.monitoring.inWorkPos),
                           commands := "Unit1.Em0.HmiInterface".cmUnwinderTopAxisB.commands,
                           interlockOk := "Unit1.Em0.ControlNodes".cm.Interlock.unwinderTopAxisB.source.posAbsolute,
                           intOut := "Unit1.Em0.HmiInterface".intCondition.Axis_01.Position.intOut);
   #_w1 := NOT (NOT #FALSE) AND "Unit1.Em0.ControlNodes".cm.Interlock.unwinderTopAxisB.source.posAbsolute[3];
   IF #_w1 THEN "Unit1.Em0.ControlNodes".cmUnwinderTopAxisB.commands.selectSetPosition := 3; END_IF;
   "Unit1.Em0.ControlNodes".cm.command.unwinderTopAxisB.posAbsolute[3] := #_w1;
END_REGION

REGION Network 43: CmUnwinderTopAxisB Position Absolute Position4
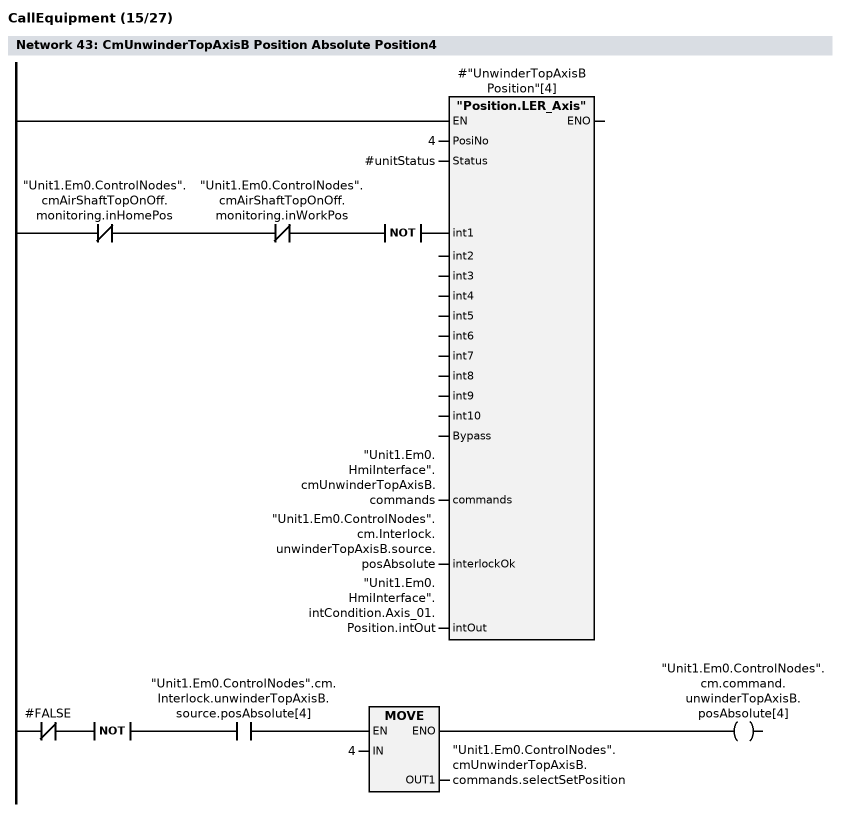
   RUNG wire#powerrail
      #"UnwinderTopAxisB Position"[4](int1 := wire#w1, PosiNo := 4, Status := #unitStatus, int2 :=, int3 :=, int4 :=, int5 :=, int6 :=, int7 :=, int8 :=, int9 :=, int10 :=, Bypass :=, commands := "Unit1.Em0.HmiInterface".cmUnwinderTopAxisB.commands, interlockOk := "Unit1.Em0.ControlNodes".cm.Interlock.unwinderTopAxisB.source.posAbsolute, intOut := "Unit1.Em0.HmiInterface".intCondition.Axis_01.Position.intOut)
   END_RUNG
   RUNG wire#powerrail
      I_Contact( "Unit1.Em0.ControlNodes".cmAirShaftTopOnOff.monitoring.inHomePos )
      I_Contact( "Unit1.Em0.ControlNodes".cmAirShaftTopOnOff.monitoring.inWorkPos )
      Not()
   END_RUNG wire#w1
   RUNG wire#powerrail
      I_Contact( #FALSE )
      Not()
      Contact( "Unit1.Em0.ControlNodes".cm.Interlock.unwinderTopAxisB.source.posAbsolute[4] )
      Move(in := 4, out1 => "Unit1.Em0.ControlNodes".cmUnwinderTopAxisB.commands.selectSetPosition)
      Coil( "Unit1.Em0.ControlNodes".cm.command.unwinderTopAxisB.posAbsolute[4] )
   END_RUNG
   // the same network as SCL:
   #"UnwinderTopAxisB Position"[4](PosiNo := 4,   // "Position.LER_Axis"
                           Status := #unitStatus,
                           int1 := NOT (NOT "Unit1.Em0.ControlNodes".cmAirShaftTopOnOff.monitoring.inHomePos AND NOT "Unit1.Em0.ControlNodes".cmAirShaftTopOnOff.monitoring.inWorkPos),
                           commands := "Unit1.Em0.HmiInterface".cmUnwinderTopAxisB.commands,
                           interlockOk := "Unit1.Em0.ControlNodes".cm.Interlock.unwinderTopAxisB.source.posAbsolute,
                           intOut := "Unit1.Em0.HmiInterface".intCondition.Axis_01.Position.intOut);
   #_w1 := NOT (NOT #FALSE) AND "Unit1.Em0.ControlNodes".cm.Interlock.unwinderTopAxisB.source.posAbsolute[4];
   IF #_w1 THEN "Unit1.Em0.ControlNodes".cmUnwinderTopAxisB.commands.selectSetPosition := 4; END_IF;
   "Unit1.Em0.ControlNodes".cm.command.unwinderTopAxisB.posAbsolute[4] := #_w1;
END_REGION

REGION Network 44: CmUnwinderTopAxisB Position Absolute Position5
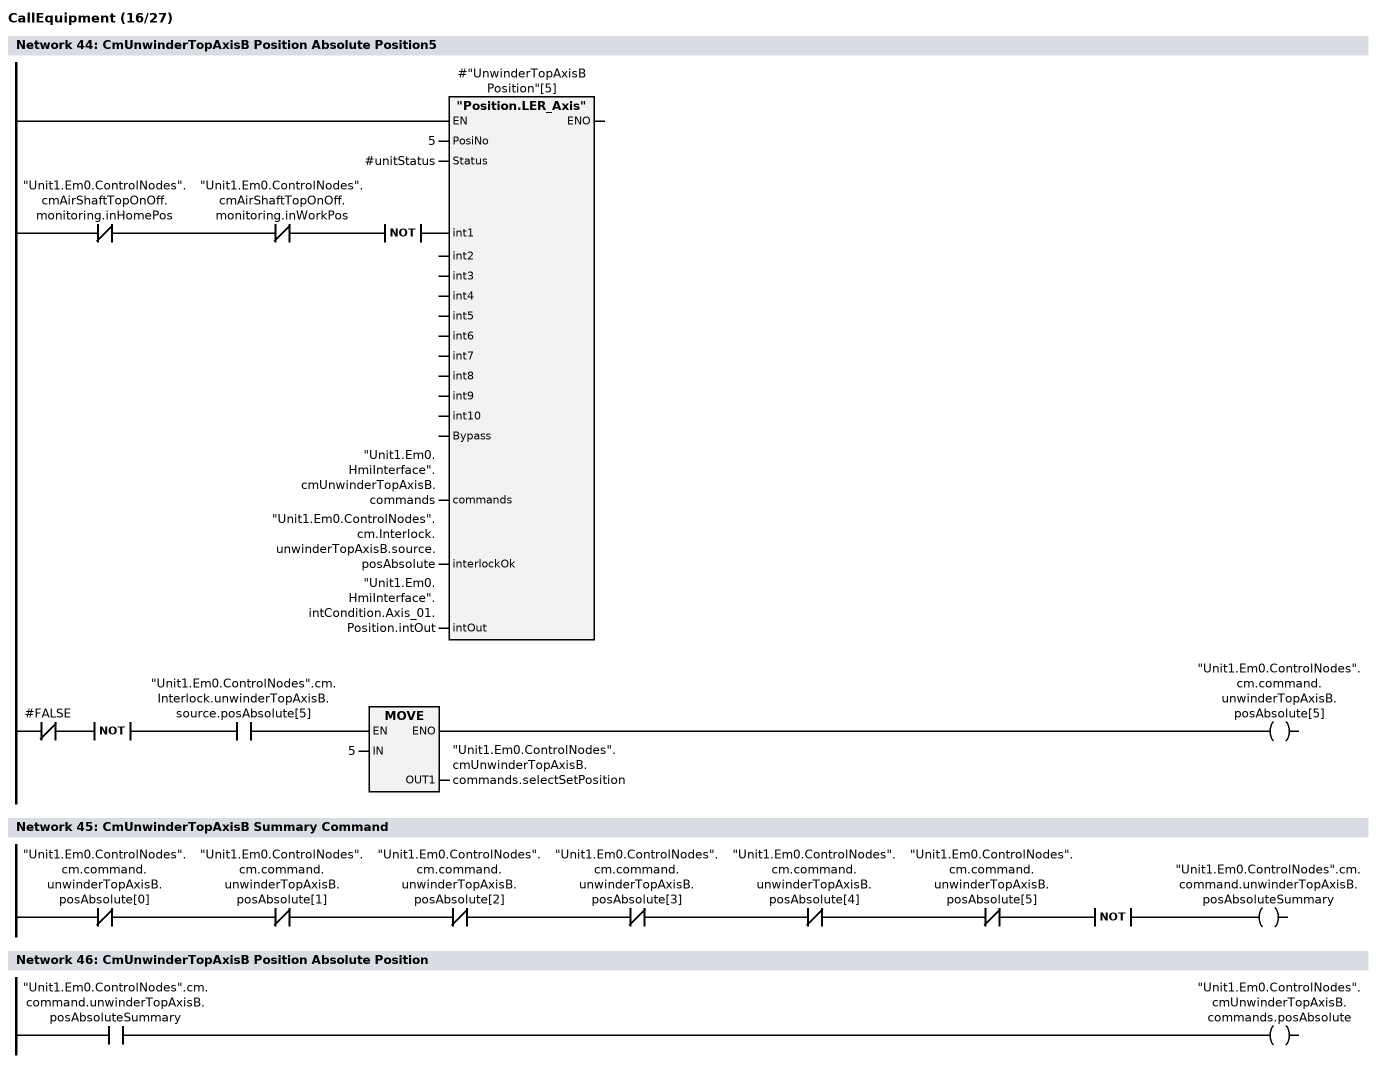
   RUNG wire#powerrail
      #"UnwinderTopAxisB Position"[5](int1 := wire#w1, PosiNo := 5, Status := #unitStatus, int2 :=, int3 :=, int4 :=, int5 :=, int6 :=, int7 :=, int8 :=, int9 :=, int10 :=, Bypass :=, commands := "Unit1.Em0.HmiInterface".cmUnwinderTopAxisB.commands, interlockOk := "Unit1.Em0.ControlNodes".cm.Interlock.unwinderTopAxisB.source.posAbsolute, intOut := "Unit1.Em0.HmiInterface".intCondition.Axis_01.Position.intOut)
   END_RUNG
   RUNG wire#powerrail
      I_Contact( "Unit1.Em0.ControlNodes".cmAirShaftTopOnOff.monitoring.inHomePos )
      I_Contact( "Unit1.Em0.ControlNodes".cmAirShaftTopOnOff.monitoring.inWorkPos )
      Not()
   END_RUNG wire#w1
   RUNG wire#powerrail
      I_Contact( #FALSE )
      Not()
      Contact( "Unit1.Em0.ControlNodes".cm.Interlock.unwinderTopAxisB.source.posAbsolute[5] )
      Move(in := 5, out1 => "Unit1.Em0.ControlNodes".cmUnwinderTopAxisB.commands.selectSetPosition)
      Coil( "Unit1.Em0.ControlNodes".cm.command.unwinderTopAxisB.posAbsolute[5] )
   END_RUNG
   // the same network as SCL:
   #"UnwinderTopAxisB Position"[5](PosiNo := 5,   // "Position.LER_Axis"
                           Status := #unitStatus,
                           int1 := NOT (NOT "Unit1.Em0.ControlNodes".cmAirShaftTopOnOff.monitoring.inHomePos AND NOT "Unit1.Em0.ControlNodes".cmAirShaftTopOnOff.monitoring.inWorkPos),
                           commands := "Unit1.Em0.HmiInterface".cmUnwinderTopAxisB.commands,
                           interlockOk := "Unit1.Em0.ControlNodes".cm.Interlock.unwinderTopAxisB.source.posAbsolute,
                           intOut := "Unit1.Em0.HmiInterface".intCondition.Axis_01.Position.intOut);
   #_w1 := NOT (NOT #FALSE) AND "Unit1.Em0.ControlNodes".cm.Interlock.unwinderTopAxisB.source.posAbsolute[5];
   IF #_w1 THEN "Unit1.Em0.ControlNodes".cmUnwinderTopAxisB.commands.selectSetPosition := 5; END_IF;
   "Unit1.Em0.ControlNodes".cm.command.unwinderTopAxisB.posAbsolute[5] := #_w1;
END_REGION

REGION Network 45: CmUnwinderTopAxisB Summary Command
   RUNG wire#powerrail
      I_Contact( "Unit1.Em0.ControlNodes".cm.command.unwinderTopAxisB.posAbsolute[0] )
      I_Contact( "Unit1.Em0.ControlNodes".cm.command.unwinderTopAxisB.posAbsolute[1] )
      I_Contact( "Unit1.Em0.ControlNodes".cm.command.unwinderTopAxisB.posAbsolute[2] )
      I_Contact( "Unit1.Em0.ControlNodes".cm.command.unwinderTopAxisB.posAbsolute[3] )
      I_Contact( "Unit1.Em0.ControlNodes".cm.command.unwinderTopAxisB.posAbsolute[4] )
      I_Contact( "Unit1.Em0.ControlNodes".cm.command.unwinderTopAxisB.posAbsolute[5] )
      Not()
      Coil( "Unit1.Em0.ControlNodes".cm.command.unwinderTopAxisB.posAbsoluteSummary )
   END_RUNG
   // the same network as SCL:
   "Unit1.Em0.ControlNodes".cm.command.unwinderTopAxisB.posAbsoluteSummary := NOT (NOT "Unit1.Em0.ControlNodes".cm.command.unwinderTopAxisB.posAbsolute[0] AND NOT "Unit1.Em0.ControlNodes".cm.command.unwinderTopAxisB.posAbsolute[1] AND NOT "Unit1.Em0.ControlNodes".cm.command.unwinderTopAxisB.posAbsolute[2] AND NOT "Unit1.Em0.ControlNodes".cm.command.unwinderTopAxisB.posAbsolute[3] AND NOT "Unit1.Em0.ControlNodes".cm.command.unwinderTopAxisB.posAbsolute[4] AND NOT "Unit1.Em0.ControlNodes".cm.command.unwinderTopAxisB.posAbsolute[5]);
END_REGION

REGION Network 46: CmUnwinderTopAxisB Position Absolute Position
   RUNG wire#powerrail
      Contact( "Unit1.Em0.ControlNodes".cm.command.unwinderTopAxisB.posAbsoluteSummary )
      Coil( "Unit1.Em0.ControlNodes".cmUnwinderTopAxisB.commands.posAbsolute )
   END_RUNG
   // the same network as SCL:
   "Unit1.Em0.ControlNodes".cmUnwinderTopAxisB.commands.posAbsolute := "Unit1.Em0.ControlNodes".cm.command.unwinderTopAxisB.posAbsoluteSummary;
END_REGION

REGION Network 47: CmUnwinderTopAxisB velocity/speed
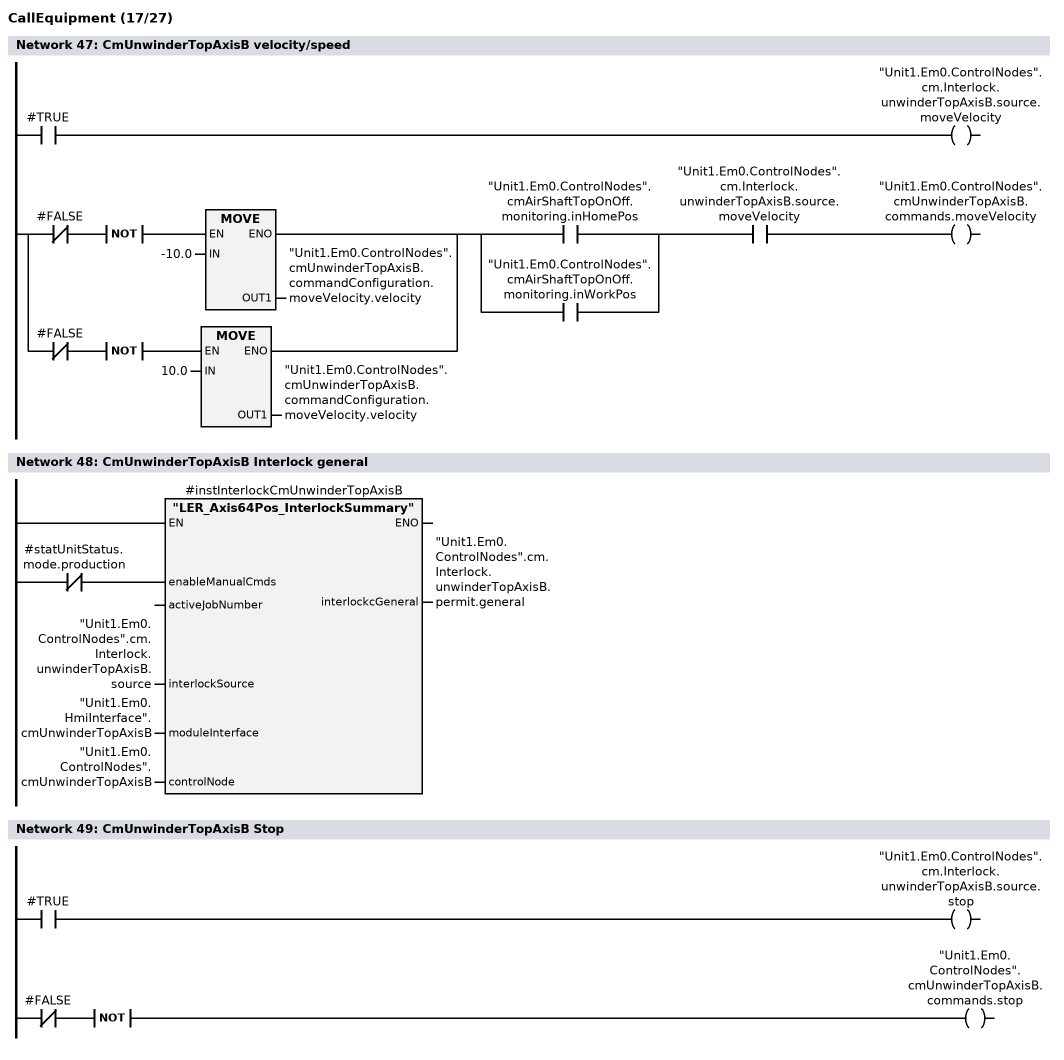
   RUNG wire#powerrail
      Contact( #TRUE )
      Coil( "Unit1.Em0.ControlNodes".cm.Interlock.unwinderTopAxisB.source.moveVelocity )
   END_RUNG
   RUNG wire#powerrail
      I_Contact( #FALSE )
      Not()
      Move(in := -10.0, out1 => "Unit1.Em0.ControlNodes".cmUnwinderTopAxisB.commandConfiguration.moveVelocity.velocity)
      wire#w1
      Contact( "Unit1.Em0.ControlNodes".cmAirShaftTopOnOff.monitoring.inHomePos )
      wire#w2
      Contact( "Unit1.Em0.ControlNodes".cm.Interlock.unwinderTopAxisB.source.moveVelocity )
      Coil( "Unit1.Em0.ControlNodes".cmUnwinderTopAxisB.commands.moveVelocity )
   END_RUNG
   RUNG wire#powerrail
      I_Contact( #FALSE )
      Not()
      Move(in := 10.0, out1 => "Unit1.Em0.ControlNodes".cmUnwinderTopAxisB.commandConfiguration.moveVelocity.velocity)
   END_RUNG wire#w1
   RUNG wire#w1
      Contact( "Unit1.Em0.ControlNodes".cmAirShaftTopOnOff.monitoring.inWorkPos )
   END_RUNG wire#w2
   // the same network as SCL:
   "Unit1.Em0.ControlNodes".cm.Interlock.unwinderTopAxisB.source.moveVelocity := #TRUE;
   IF NOT (NOT #FALSE) THEN
       "Unit1.Em0.ControlNodes".cmUnwinderTopAxisB.commandConfiguration.moveVelocity.velocity := -10.0;
       "Unit1.Em0.ControlNodes".cmUnwinderTopAxisB.commandConfiguration.moveVelocity.velocity := 10.0;
   END_IF;
   "Unit1.Em0.ControlNodes".cmUnwinderTopAxisB.commands.moveVelocity := (NOT (NOT #FALSE) OR NOT (NOT #FALSE)) AND ("Unit1.Em0.ControlNodes".cmAirShaftTopOnOff.monitoring.inHomePos OR "Unit1.Em0.ControlNodes".cmAirShaftTopOnOff.monitoring.inWorkPos) AND "Unit1.Em0.ControlNodes".cm.Interlock.unwinderTopAxisB.source.moveVelocity;
END_REGION

REGION Network 48: CmUnwinderTopAxisB Interlock general
   RUNG wire#powerrail
      #instInterlockCmUnwinderTopAxisB(enableManualCmds := wire#w1, activeJobNumber :=, interlockSource := "Unit1.Em0.ControlNodes".cm.Interlock.unwinderTopAxisB.source, moduleInterface := "Unit1.Em0.HmiInterface".cmUnwinderTopAxisB, controlNode := "Unit1.Em0.ControlNodes".cmUnwinderTopAxisB, interlockcGeneral => "Unit1.Em0.ControlNodes".cm.Interlock.unwinderTopAxisB.permit.general)
   END_RUNG
   RUNG wire#powerrail
      I_Contact( #statUnitStatus.mode.production )
   END_RUNG wire#w1
   // the same network as SCL:
   #instInterlockCmUnwinderTopAxisB(enableManualCmds := NOT #statUnitStatus.mode.production,   // "LER_Axis64Pos_InterlockSummary"
                           interlockSource := "Unit1.Em0.ControlNodes".cm.Interlock.unwinderTopAxisB.source,
                           moduleInterface := "Unit1.Em0.HmiInterface".cmUnwinderTopAxisB,
                           controlNode := "Unit1.Em0.ControlNodes".cmUnwinderTopAxisB,
                           interlockcGeneral => "Unit1.Em0.ControlNodes".cm.Interlock.unwinderTopAxisB.permit.general);
END_REGION

REGION Network 49: CmUnwinderTopAxisB Stop
   RUNG wire#powerrail
      Contact( #TRUE )
      Coil( "Unit1.Em0.ControlNodes".cm.Interlock.unwinderTopAxisB.source.stop )
   END_RUNG
   RUNG wire#powerrail
      I_Contact( #FALSE )
      Not()
      Coil( "Unit1.Em0.ControlNodes".cmUnwinderTopAxisB.commands.stop )
   END_RUNG
   // the same network as SCL:
   "Unit1.Em0.ControlNodes".cm.Interlock.unwinderTopAxisB.source.stop := #TRUE;
   "Unit1.Em0.ControlNodes".cmUnwinderTopAxisB.commands.stop := NOT (NOT #FALSE);
END_REGION

REGION Network 50: Cm Unwinder Top AxisB FB Call
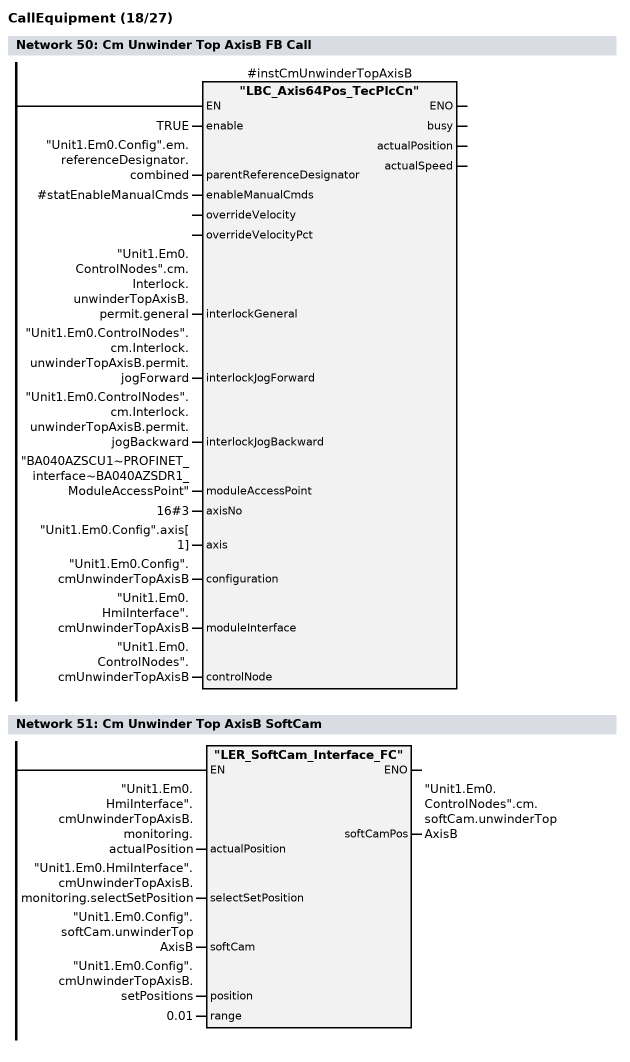
   RUNG wire#powerrail
      #instCmUnwinderTopAxisB(enable := TRUE, parentReferenceDesignator := "Unit1.Em0.Config".em.referenceDesignator.combined, enableManualCmds := #statEnableManualCmds, overrideVelocity :=, overrideVelocityPct :=, interlockGeneral := "Unit1.Em0.ControlNodes".cm.Interlock.unwinderTopAxisB.permit.general, interlockJogForward := "Unit1.Em0.ControlNodes".cm.Interlock.unwinderTopAxisB.permit.jogForward, interlockJogBackward := "Unit1.Em0.ControlNodes".cm.Interlock.unwinderTopAxisB.permit.jogBackward, moduleAccessPoint := "BA040AZSCU1~PROFINET_interface~BA040AZSDR1_ModuleAccessPoint", axisNo := 16#3, axis := "Unit1.Em0.Config".axis[1], configuration := "Unit1.Em0.Config".cmUnwinderTopAxisB, moduleInterface := "Unit1.Em0.HmiInterface".cmUnwinderTopAxisB, controlNode := "Unit1.Em0.ControlNodes".cmUnwinderTopAxisB, busy =>, actualPosition =>, actualSpeed =>)
   END_RUNG
   // the same network as SCL:
   #instCmUnwinderTopAxisB(enable := TRUE,   // "LBC_Axis64Pos_TecPlcCn"
                           parentReferenceDesignator := "Unit1.Em0.Config".em.referenceDesignator.combined,
                           enableManualCmds := #statEnableManualCmds,
                           interlockGeneral := "Unit1.Em0.ControlNodes".cm.Interlock.unwinderTopAxisB.permit.general,
                           interlockJogForward := "Unit1.Em0.ControlNodes".cm.Interlock.unwinderTopAxisB.permit.jogForward,
                           interlockJogBackward := "Unit1.Em0.ControlNodes".cm.Interlock.unwinderTopAxisB.permit.jogBackward,
                           moduleAccessPoint := "BA040AZSCU1~PROFINET_interface~BA040AZSDR1_ModuleAccessPoint",
                           axisNo := 16#3,
                           axis := "Unit1.Em0.Config".axis[1],
                           configuration := "Unit1.Em0.Config".cmUnwinderTopAxisB,
                           moduleInterface := "Unit1.Em0.HmiInterface".cmUnwinderTopAxisB,
                           controlNode := "Unit1.Em0.ControlNodes".cmUnwinderTopAxisB);
END_REGION

REGION Network 51: Cm Unwinder Top AxisB SoftCam
   RUNG wire#powerrail
      "LER_SoftCam_Interface_FC"(actualPosition := "Unit1.Em0.HmiInterface".cmUnwinderTopAxisB.monitoring.actualPosition, selectSetPosition := "Unit1.Em0.HmiInterface".cmUnwinderTopAxisB.monitoring.selectSetPosition, softCam := "Unit1.Em0.Config".softCam.unwinderTopAxisB, position := "Unit1.Em0.Config".cmUnwinderTopAxisB.setPositions, range := 0.01, softCamPos => "Unit1.Em0.ControlNodes".cm.softCam.unwinderTopAxisB)
   END_RUNG
   // the same network as SCL:
   "LER_SoftCam_Interface_FC"(actualPosition := "Unit1.Em0.HmiInterface".cmUnwinderTopAxisB.monitoring.actualPosition,
                           selectSetPosition := "Unit1.Em0.HmiInterface".cmUnwinderTopAxisB.monitoring.selectSetPosition,
                           softCam := "Unit1.Em0.Config".softCam.unwinderTopAxisB,
                           position := "Unit1.Em0.Config".cmUnwinderTopAxisB.setPositions,
                           range := 0.01,
                           softCamPos => "Unit1.Em0.ControlNodes".cm.softCam.unwinderTopAxisB);
END_REGION

REGION Network 52: *************** Servo Torque Calculation (Axis) *******************
END_REGION

REGION Network 53: Call instCmUnwinderTopAxisB Torque Cal
END_REGION

REGION Network 54: ******************** Brake Test (Axis) ********************
END_REGION

REGION Network 55: Unwinder Top B-Axis Brake Test
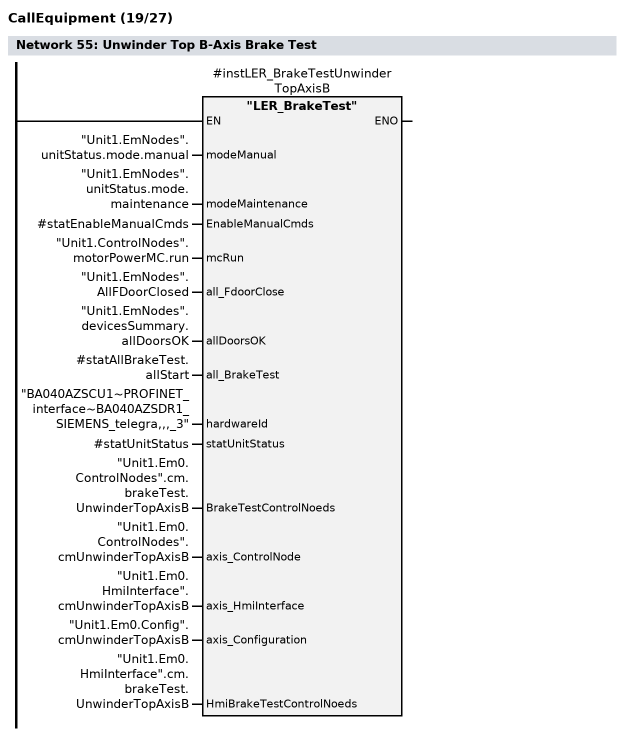
   RUNG wire#powerrail
      #instLER_BrakeTestUnwinderTopAxisB(modeManual := "Unit1.EmNodes".unitStatus.mode.manual, modeMaintenance := "Unit1.EmNodes".unitStatus.mode.maintenance, EnableManualCmds := #statEnableManualCmds, mcRun := "Unit1.ControlNodes".motorPowerMC.run, all_FdoorClose := "Unit1.EmNodes".AllFDoorClosed, allDoorsOK := "Unit1.EmNodes".devicesSummary.allDoorsOK, all_BrakeTest := #statAllBrakeTest.allStart, hardwareId := "BA040AZSCU1~PROFINET_interface~BA040AZSDR1_SIEMENS_telegra,,,_3", statUnitStatus := #statUnitStatus, BrakeTestControlNoeds := "Unit1.Em0.ControlNodes".cm.brakeTest.UnwinderTopAxisB, axis_ControlNode := "Unit1.Em0.ControlNodes".cmUnwinderTopAxisB, axis_HmiInterface := "Unit1.Em0.HmiInterface".cmUnwinderTopAxisB, axis_Configuration := "Unit1.Em0.Config".cmUnwinderTopAxisB, HmiBrakeTestControlNoeds := "Unit1.Em0.HmiInterface".cm.brakeTest.UnwinderTopAxisB)
   END_RUNG
   // the same network as SCL:
   #instLER_BrakeTestUnwinderTopAxisB(modeManual := "Unit1.EmNodes".unitStatus.mode.manual,   // "LER_BrakeTest"
                           modeMaintenance := "Unit1.EmNodes".unitStatus.mode.maintenance,
                           EnableManualCmds := #statEnableManualCmds,
                           mcRun := "Unit1.ControlNodes".motorPowerMC.run,
                           all_FdoorClose := "Unit1.EmNodes".AllFDoorClosed,
                           allDoorsOK := "Unit1.EmNodes".devicesSummary.allDoorsOK,
                           all_BrakeTest := #statAllBrakeTest.allStart,
                           hardwareId := "BA040AZSCU1~PROFINET_interface~BA040AZSDR1_SIEMENS_telegra,,,_3",
                           statUnitStatus := #statUnitStatus,
                           BrakeTestControlNoeds := "Unit1.Em0.ControlNodes".cm.brakeTest.UnwinderTopAxisB,
                           axis_ControlNode := "Unit1.Em0.ControlNodes".cmUnwinderTopAxisB,
                           axis_HmiInterface := "Unit1.Em0.HmiInterface".cmUnwinderTopAxisB,
                           axis_Configuration := "Unit1.Em0.Config".cmUnwinderTopAxisB,
                           HmiBrakeTestControlNoeds := "Unit1.Em0.HmiInterface".cm.brakeTest.UnwinderTopAxisB);
END_REGION

REGION Network 56: ********** Control Modules (TwoWayActuator) **********
END_REGION

REGION Network 57: Reset CMS
   // Reset Axis when the unit is in the resetting state.
END_REGION

REGION Network 59: CmUnwinderAirShaftTop On
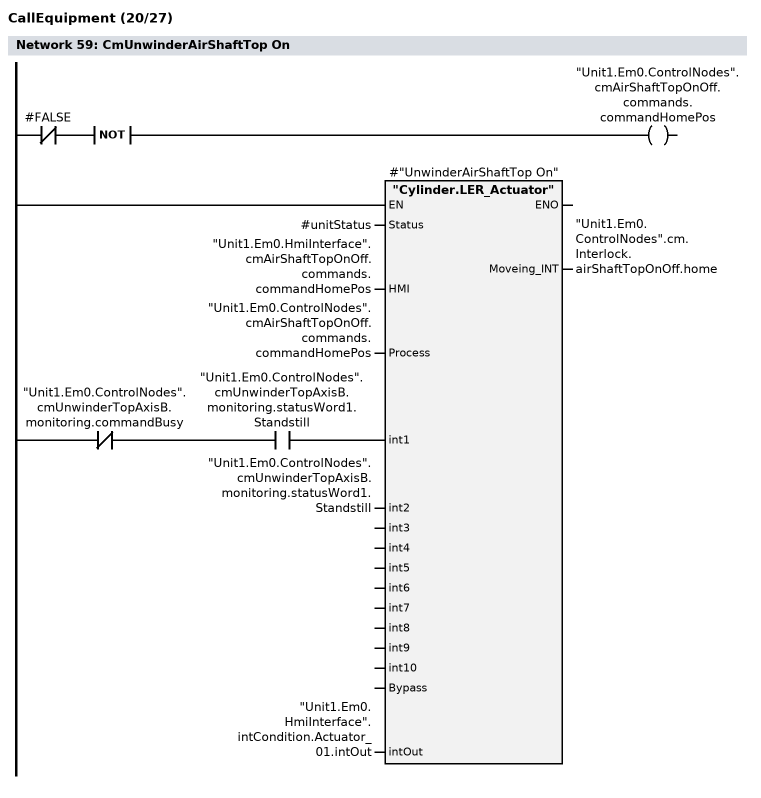
   RUNG wire#powerrail
      I_Contact( #FALSE )
      Not()
      Coil( "Unit1.Em0.ControlNodes".cmAirShaftTopOnOff.commands.commandHomePos )
   END_RUNG
   RUNG wire#powerrail
      #"UnwinderAirShaftTop On"(int1 := wire#w1, Status := #unitStatus, HMI := "Unit1.Em0.HmiInterface".cmAirShaftTopOnOff.commands.commandHomePos, Process := "Unit1.Em0.ControlNodes".cmAirShaftTopOnOff.commands.commandHomePos, int2 := "Unit1.Em0.ControlNodes".cmUnwinderTopAxisB.monitoring.statusWord1.Standstill, int3 :=, int4 :=, int5 :=, int6 :=, int7 :=, int8 :=, int9 :=, int10 :=, Bypass :=, intOut := "Unit1.Em0.HmiInterface".intCondition.Actuator_01.intOut, Moveing_INT => "Unit1.Em0.ControlNodes".cm.Interlock.airShaftTopOnOff.home)
   END_RUNG
   RUNG wire#powerrail
      I_Contact( "Unit1.Em0.ControlNodes".cmUnwinderTopAxisB.monitoring.commandBusy )
      Contact( "Unit1.Em0.ControlNodes".cmUnwinderTopAxisB.monitoring.statusWord1.Standstill )
   END_RUNG wire#w1
   // the same network as SCL:
   "Unit1.Em0.ControlNodes".cmAirShaftTopOnOff.commands.commandHomePos := NOT (NOT #FALSE);
   #"UnwinderAirShaftTop On"(Status := #unitStatus,   // "Cylinder.LER_Actuator"
                           HMI := "Unit1.Em0.HmiInterface".cmAirShaftTopOnOff.commands.commandHomePos,
                           Process := "Unit1.Em0.ControlNodes".cmAirShaftTopOnOff.commands.commandHomePos,
                           int1 := NOT "Unit1.Em0.ControlNodes".cmUnwinderTopAxisB.monitoring.commandBusy AND "Unit1.Em0.ControlNodes".cmUnwinderTopAxisB.monitoring.statusWord1.Standstill,
                           int2 := "Unit1.Em0.ControlNodes".cmUnwinderTopAxisB.monitoring.statusWord1.Standstill,
                           intOut := "Unit1.Em0.HmiInterface".intCondition.Actuator_01.intOut,
                           Moveing_INT => "Unit1.Em0.ControlNodes".cm.Interlock.airShaftTopOnOff.home);
END_REGION

REGION Network 60: CmUnwinderAirShaftTop Off
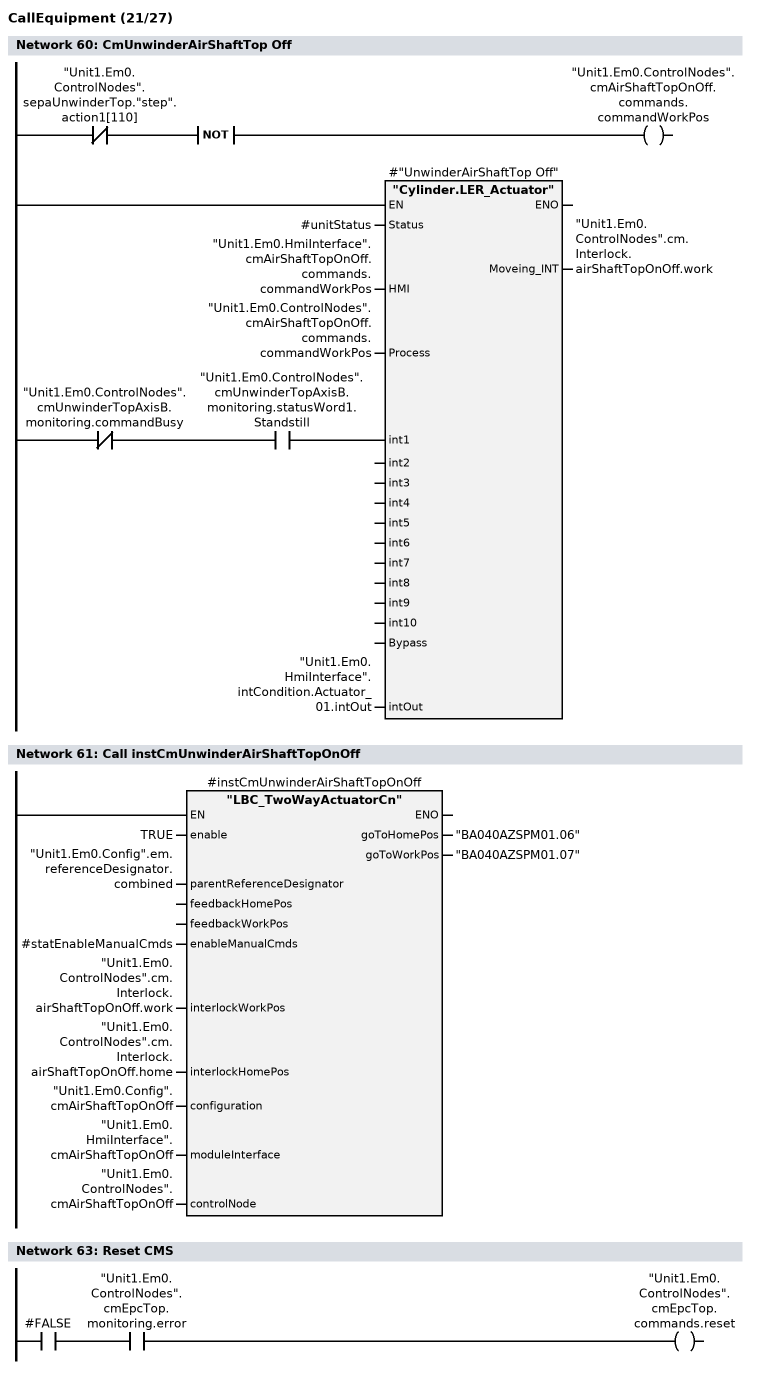
   RUNG wire#powerrail
      I_Contact( "Unit1.Em0.ControlNodes".sepaUnwinderTop."step".action1[110] )
      Not()
      Coil( "Unit1.Em0.ControlNodes".cmAirShaftTopOnOff.commands.commandWorkPos )
   END_RUNG
   RUNG wire#powerrail
      #"UnwinderAirShaftTop Off"(int1 := wire#w1, Status := #unitStatus, HMI := "Unit1.Em0.HmiInterface".cmAirShaftTopOnOff.commands.commandWorkPos, Process := "Unit1.Em0.ControlNodes".cmAirShaftTopOnOff.commands.commandWorkPos, int2 :=, int3 :=, int4 :=, int5 :=, int6 :=, int7 :=, int8 :=, int9 :=, int10 :=, Bypass :=, intOut := "Unit1.Em0.HmiInterface".intCondition.Actuator_01.intOut, Moveing_INT => "Unit1.Em0.ControlNodes".cm.Interlock.airShaftTopOnOff.work)
   END_RUNG
   RUNG wire#powerrail
      I_Contact( "Unit1.Em0.ControlNodes".cmUnwinderTopAxisB.monitoring.commandBusy )
      Contact( "Unit1.Em0.ControlNodes".cmUnwinderTopAxisB.monitoring.statusWord1.Standstill )
   END_RUNG wire#w1
   // the same network as SCL:
   "Unit1.Em0.ControlNodes".cmAirShaftTopOnOff.commands.commandWorkPos := NOT (NOT "Unit1.Em0.ControlNodes".sepaUnwinderTop."step".action1[110]);
   #"UnwinderAirShaftTop Off"(Status := #unitStatus,   // "Cylinder.LER_Actuator"
                           HMI := "Unit1.Em0.HmiInterface".cmAirShaftTopOnOff.commands.commandWorkPos,
                           Process := "Unit1.Em0.ControlNodes".cmAirShaftTopOnOff.commands.commandWorkPos,
                           int1 := NOT "Unit1.Em0.ControlNodes".cmUnwinderTopAxisB.monitoring.commandBusy AND "Unit1.Em0.ControlNodes".cmUnwinderTopAxisB.monitoring.statusWord1.Standstill,
                           intOut := "Unit1.Em0.HmiInterface".intCondition.Actuator_01.intOut,
                           Moveing_INT => "Unit1.Em0.ControlNodes".cm.Interlock.airShaftTopOnOff.work);
END_REGION

REGION Network 61: Call instCmUnwinderAirShaftTopOnOff
   RUNG wire#powerrail
      #instCmUnwinderAirShaftTopOnOff(enable := TRUE, parentReferenceDesignator := "Unit1.Em0.Config".em.referenceDesignator.combined, feedbackHomePos :=, feedbackWorkPos :=, enableManualCmds := #statEnableManualCmds, interlockWorkPos := "Unit1.Em0.ControlNodes".cm.Interlock.airShaftTopOnOff.work, interlockHomePos := "Unit1.Em0.ControlNodes".cm.Interlock.airShaftTopOnOff.home, configuration := "Unit1.Em0.Config".cmAirShaftTopOnOff, moduleInterface := "Unit1.Em0.HmiInterface".cmAirShaftTopOnOff, controlNode := "Unit1.Em0.ControlNodes".cmAirShaftTopOnOff, goToHomePos => "BA040AZSPM01.06", goToWorkPos => "BA040AZSPM01.07")
   END_RUNG
   // the same network as SCL:
   #instCmUnwinderAirShaftTopOnOff(enable := TRUE,   // "LBC_TwoWayActuatorCn"
                           parentReferenceDesignator := "Unit1.Em0.Config".em.referenceDesignator.combined,
                           enableManualCmds := #statEnableManualCmds,
                           interlockWorkPos := "Unit1.Em0.ControlNodes".cm.Interlock.airShaftTopOnOff.work,
                           interlockHomePos := "Unit1.Em0.ControlNodes".cm.Interlock.airShaftTopOnOff.home,
                           configuration := "Unit1.Em0.Config".cmAirShaftTopOnOff,
                           moduleInterface := "Unit1.Em0.HmiInterface".cmAirShaftTopOnOff,
                           controlNode := "Unit1.Em0.ControlNodes".cmAirShaftTopOnOff,
                           goToHomePos => "BA040AZSPM01.06",
                           goToWorkPos => "BA040AZSPM01.07");
END_REGION

REGION Network 62: ******************** Control Modules (Accessories) ********************
END_REGION

REGION Network 63: Reset CMS
   RUNG wire#powerrail
      Contact( #FALSE )
      Contact( "Unit1.Em0.ControlNodes".cmEpcTop.monitoring.error )
      Coil( "Unit1.Em0.ControlNodes".cmEpcTop.commands.reset )
   END_RUNG
   // the same network as SCL:
   "Unit1.Em0.ControlNodes".cmEpcTop.commands.reset := #FALSE AND "Unit1.Em0.ControlNodes".cmEpcTop.monitoring.error;
END_REGION

REGION Network 64: CmUnwinderTopEpcControllerInterface Interlock
END_REGION

REGION Network 65: CmUnwinderTopEpcControllerInterface Commands
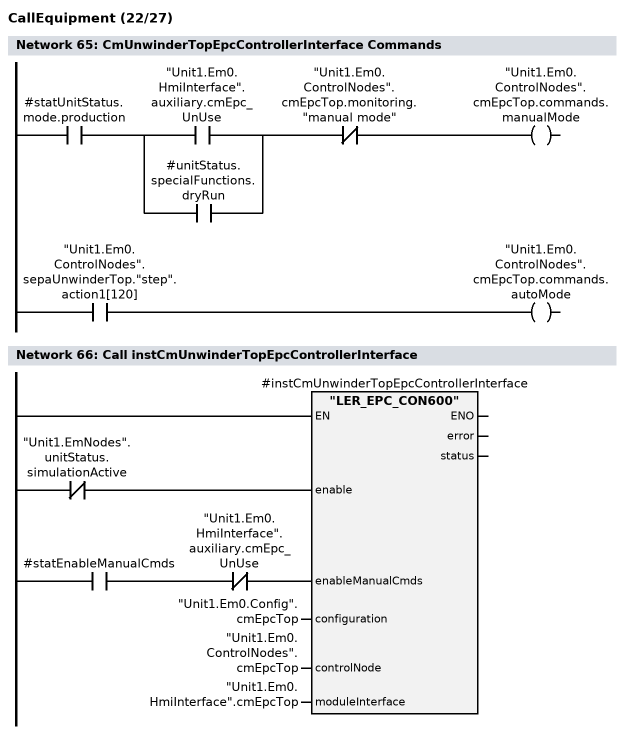
   RUNG wire#powerrail
      Contact( #statUnitStatus.mode.production )
      wire#w1
      Contact( "Unit1.Em0.HmiInterface".auxiliary.cmEpc_UnUse )
      wire#w2
      I_Contact( "Unit1.Em0.ControlNodes".cmEpcTop.monitoring."manual mode" )
      Coil( "Unit1.Em0.ControlNodes".cmEpcTop.commands.manualMode )
   END_RUNG
   RUNG wire#w1
      Contact( #unitStatus.specialFunctions.dryRun )
   END_RUNG wire#w2
   RUNG wire#powerrail
      Contact( "Unit1.Em0.ControlNodes".sepaUnwinderTop."step".action1[120] )
      Coil( "Unit1.Em0.ControlNodes".cmEpcTop.commands.autoMode )
   END_RUNG
   // the same network as SCL:
   "Unit1.Em0.ControlNodes".cmEpcTop.commands.manualMode := #statUnitStatus.mode.production AND ("Unit1.Em0.HmiInterface".auxiliary.cmEpc_UnUse OR #unitStatus.specialFunctions.dryRun) AND NOT "Unit1.Em0.ControlNodes".cmEpcTop.monitoring."manual mode";
   "Unit1.Em0.ControlNodes".cmEpcTop.commands.autoMode := "Unit1.Em0.ControlNodes".sepaUnwinderTop."step".action1[120];
END_REGION

REGION Network 66: Call instCmUnwinderTopEpcControllerInterface
   RUNG wire#powerrail
      #instCmUnwinderTopEpcControllerInterface(enable := wire#w1, enableManualCmds := wire#w2, configuration := "Unit1.Em0.Config".cmEpcTop, controlNode := "Unit1.Em0.ControlNodes".cmEpcTop, moduleInterface := "Unit1.Em0.HmiInterface".cmEpcTop, error =>, status =>)
   END_RUNG
   RUNG wire#powerrail
      I_Contact( "Unit1.EmNodes".unitStatus.simulationActive )
   END_RUNG wire#w1
   RUNG wire#powerrail
      Contact( #statEnableManualCmds )
      I_Contact( "Unit1.Em0.HmiInterface".auxiliary.cmEpc_UnUse )
   END_RUNG wire#w2
   // the same network as SCL:
   #instCmUnwinderTopEpcControllerInterface(enable := NOT "Unit1.EmNodes".unitStatus.simulationActive,   // "LER_EPC_CON600"
                           enableManualCmds := #statEnableManualCmds AND NOT "Unit1.Em0.HmiInterface".auxiliary.cmEpc_UnUse,
                           configuration := "Unit1.Em0.Config".cmEpcTop,
                           controlNode := "Unit1.Em0.ControlNodes".cmEpcTop,
                           moduleInterface := "Unit1.Em0.HmiInterface".cmEpcTop);
END_REGION

REGION Network 67: *************** Feedback to Unit ***************************
END_REGION

REGION Network 68: Determine StateComplete (SC) in Mode Production
   // Conditions for the Equipment Modules "stateComplete" feedback to the unit. This feedback is given when the task in for the respective state is complete.
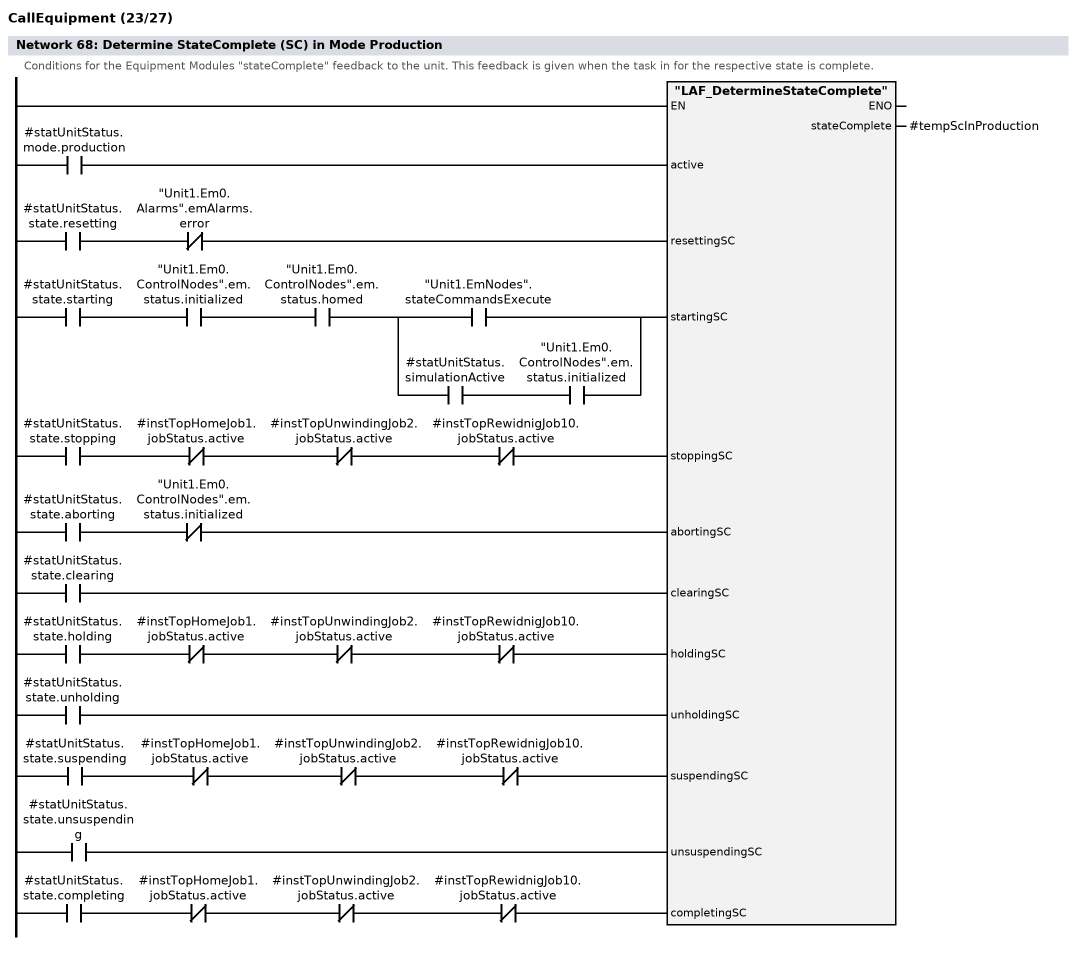
   RUNG wire#powerrail
      "LAF_DetermineStateComplete"(active := wire#w1, resettingSC := wire#w2, startingSC := wire#w4, stoppingSC := wire#w5, abortingSC := wire#w6, clearingSC := wire#w7, holdingSC := wire#w8, unholdingSC := wire#w9, suspendingSC := wire#w10, unsuspendingSC := wire#w11, completingSC := wire#w12, stateComplete => #tempScInProduction)
   END_RUNG
   RUNG wire#powerrail
      Contact( #statUnitStatus.mode.production )
   END_RUNG wire#w1
   RUNG wire#powerrail
      Contact( #statUnitStatus.state.resetting )
      I_Contact( "Unit1.Em0.Alarms".emAlarms.error )
   END_RUNG wire#w2
   RUNG wire#powerrail
      Contact( #statUnitStatus.state.starting )
      Contact( "Unit1.Em0.ControlNodes".em.status.initialized )
      Contact( "Unit1.Em0.ControlNodes".em.status.homed )
      wire#w3
      Contact( "Unit1.EmNodes".stateCommandsExecute )
   END_RUNG wire#w4
   RUNG wire#w3
      Contact( #statUnitStatus.simulationActive )
      Contact( "Unit1.Em0.ControlNodes".em.status.initialized )
   END_RUNG wire#w4
   RUNG wire#powerrail
      Contact( #statUnitStatus.state.stopping )
      I_Contact( #instTopHomeJob1.jobStatus.active )
      I_Contact( #instTopUnwindingJob2.jobStatus.active )
      I_Contact( #instTopRewidnigJob10.jobStatus.active )
   END_RUNG wire#w5
   RUNG wire#powerrail
      Contact( #statUnitStatus.state.aborting )
      I_Contact( "Unit1.Em0.ControlNodes".em.status.initialized )
   END_RUNG wire#w6
   RUNG wire#powerrail
      Contact( #statUnitStatus.state.clearing )
   END_RUNG wire#w7
   RUNG wire#powerrail
      Contact( #statUnitStatus.state.holding )
      I_Contact( #instTopHomeJob1.jobStatus.active )
      I_Contact( #instTopUnwindingJob2.jobStatus.active )
      I_Contact( #instTopRewidnigJob10.jobStatus.active )
   END_RUNG wire#w8
   RUNG wire#powerrail
      Contact( #statUnitStatus.state.unholding )
   END_RUNG wire#w9
   RUNG wire#powerrail
      Contact( #statUnitStatus.state.suspending )
      I_Contact( #instTopHomeJob1.jobStatus.active )
      I_Contact( #instTopUnwindingJob2.jobStatus.active )
      I_Contact( #instTopRewidnigJob10.jobStatus.active )
   END_RUNG wire#w10
   RUNG wire#powerrail
      Contact( #statUnitStatus.state.unsuspending )
   END_RUNG wire#w11
   RUNG wire#powerrail
      Contact( #statUnitStatus.state.completing )
      I_Contact( #instTopHomeJob1.jobStatus.active )
      I_Contact( #instTopUnwindingJob2.jobStatus.active )
      I_Contact( #instTopRewidnigJob10.jobStatus.active )
   END_RUNG wire#w12
   // the same network as SCL:
   "LAF_DetermineStateComplete"(active := #statUnitStatus.mode.production,
                           resettingSC := #statUnitStatus.state.resetting AND NOT "Unit1.Em0.Alarms".emAlarms.error,
                           startingSC := #statUnitStatus.state.starting AND "Unit1.Em0.ControlNodes".em.status.initialized AND "Unit1.Em0.ControlNodes".em.status.homed AND ("Unit1.EmNodes".stateCommandsExecute OR (#statUnitStatus.simulationActive AND "Unit1.Em0.ControlNodes".em.status.initialized)),
                           stoppingSC := #statUnitStatus.state.stopping AND NOT #instTopHomeJob1.jobStatus.active AND NOT #instTopUnwindingJob2.jobStatus.active AND NOT #instTopRewidnigJob10.jobStatus.active,
                           abortingSC := #statUnitStatus.state.aborting AND NOT "Unit1.Em0.ControlNodes".em.status.initialized,
                           clearingSC := #statUnitStatus.state.clearing,
                           holdingSC := #statUnitStatus.state.holding AND NOT #instTopHomeJob1.jobStatus.active AND NOT #instTopUnwindingJob2.jobStatus.active AND NOT #instTopRewidnigJob10.jobStatus.active,
                           unholdingSC := #statUnitStatus.state.unholding,
                           suspendingSC := #statUnitStatus.state.suspending AND NOT #instTopHomeJob1.jobStatus.active AND NOT #instTopUnwindingJob2.jobStatus.active AND NOT #instTopRewidnigJob10.jobStatus.active,
                           unsuspendingSC := #statUnitStatus.state.unsuspending,
                           completingSC := #statUnitStatus.state.completing AND NOT #instTopHomeJob1.jobStatus.active AND NOT #instTopUnwindingJob2.jobStatus.active AND NOT #instTopRewidnigJob10.jobStatus.active,
                           stateComplete => #tempScInProduction);
END_REGION

REGION Network 69: Determine StateComplete (SC) in Mode Maintenance/Manual
   // Conditions for the Equipment Modules "stateComplete" feedback to the unit. This feedback is given when the task in for the respective state is complete.
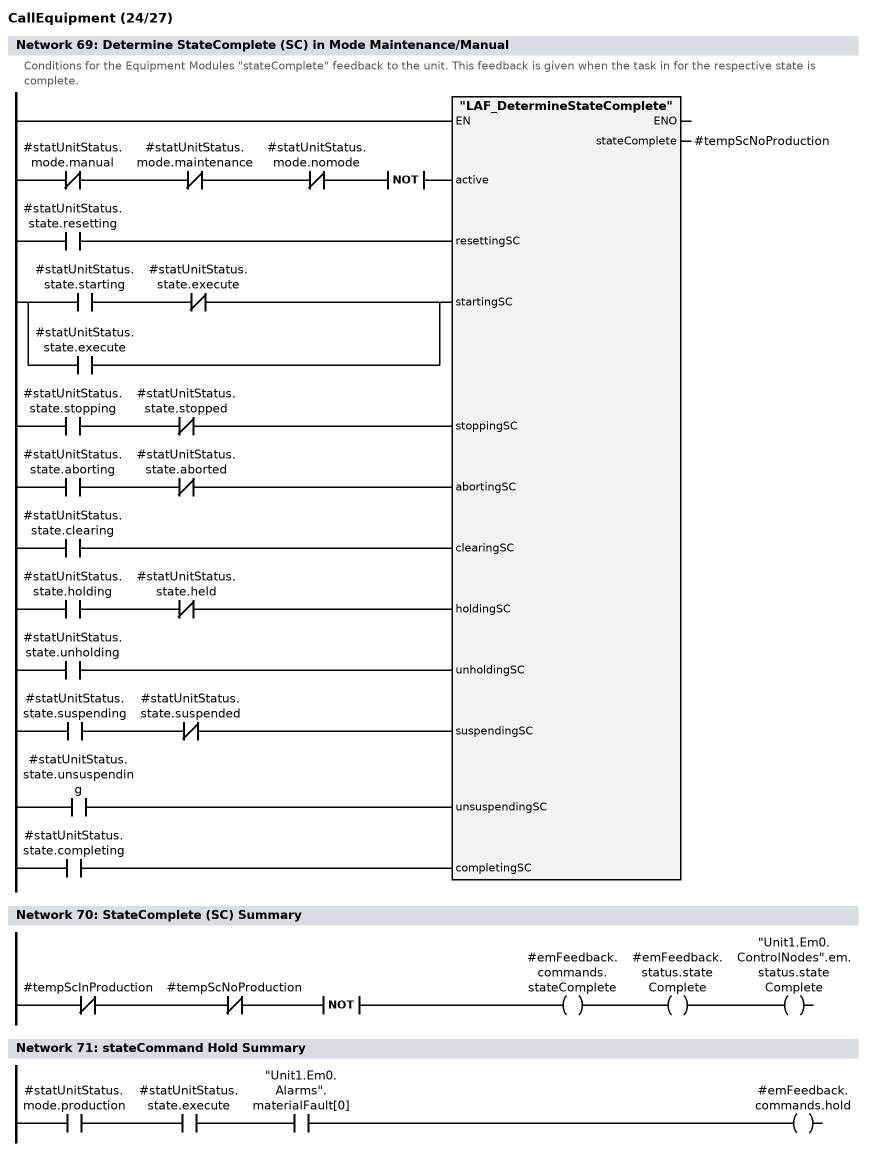
   RUNG wire#powerrail
      "LAF_DetermineStateComplete"(active := wire#w1, resettingSC := wire#w2, startingSC := wire#w3, stoppingSC := wire#w4, abortingSC := wire#w5, clearingSC := wire#w6, holdingSC := wire#w7, unholdingSC := wire#w8, suspendingSC := wire#w9, unsuspendingSC := wire#w10, completingSC := wire#w11, stateComplete => #tempScNoProduction)
   END_RUNG
   RUNG wire#powerrail
      I_Contact( #statUnitStatus.mode.manual )
      I_Contact( #statUnitStatus.mode.maintenance )
      I_Contact( #statUnitStatus.mode.nomode )
      Not()
   END_RUNG wire#w1
   RUNG wire#powerrail
      Contact( #statUnitStatus.state.resetting )
   END_RUNG wire#w2
   RUNG wire#powerrail
      Contact( #statUnitStatus.state.starting )
      I_Contact( #statUnitStatus.state.execute )
   END_RUNG wire#w3
   RUNG wire#powerrail
      Contact( #statUnitStatus.state.execute )
   END_RUNG wire#w3
   RUNG wire#powerrail
      Contact( #statUnitStatus.state.stopping )
      I_Contact( #statUnitStatus.state.stopped )
   END_RUNG wire#w4
   RUNG wire#powerrail
      Contact( #statUnitStatus.state.aborting )
      I_Contact( #statUnitStatus.state.aborted )
   END_RUNG wire#w5
   RUNG wire#powerrail
      Contact( #statUnitStatus.state.clearing )
   END_RUNG wire#w6
   RUNG wire#powerrail
      Contact( #statUnitStatus.state.holding )
      I_Contact( #statUnitStatus.state.held )
   END_RUNG wire#w7
   RUNG wire#powerrail
      Contact( #statUnitStatus.state.unholding )
   END_RUNG wire#w8
   RUNG wire#powerrail
      Contact( #statUnitStatus.state.suspending )
      I_Contact( #statUnitStatus.state.suspended )
   END_RUNG wire#w9
   RUNG wire#powerrail
      Contact( #statUnitStatus.state.unsuspending )
   END_RUNG wire#w10
   RUNG wire#powerrail
      Contact( #statUnitStatus.state.completing )
   END_RUNG wire#w11
   // the same network as SCL:
   "LAF_DetermineStateComplete"(active := NOT (NOT #statUnitStatus.mode.manual AND NOT #statUnitStatus.mode.maintenance AND NOT #statUnitStatus.mode.nomode),
                           resettingSC := #statUnitStatus.state.resetting,
                           startingSC := (#statUnitStatus.state.starting AND NOT #statUnitStatus.state.execute) OR #statUnitStatus.state.execute,
                           stoppingSC := #statUnitStatus.state.stopping AND NOT #statUnitStatus.state.stopped,
                           abortingSC := #statUnitStatus.state.aborting AND NOT #statUnitStatus.state.aborted,
                           clearingSC := #statUnitStatus.state.clearing,
                           holdingSC := #statUnitStatus.state.holding AND NOT #statUnitStatus.state.held,
                           unholdingSC := #statUnitStatus.state.unholding,
                           suspendingSC := #statUnitStatus.state.suspending AND NOT #statUnitStatus.state.suspended,
                           unsuspendingSC := #statUnitStatus.state.unsuspending,
                           completingSC := #statUnitStatus.state.completing,
                           stateComplete => #tempScNoProduction);
END_REGION

REGION Network 70: StateComplete (SC) Summary
   RUNG wire#powerrail
      I_Contact( #tempScInProduction )
      I_Contact( #tempScNoProduction )
      Not()
      Coil( #emFeedback.commands.stateComplete )
      Coil( #emFeedback.status.stateComplete )
      Coil( "Unit1.Em0.ControlNodes".em.status.stateComplete )
   END_RUNG
   // the same network as SCL:
   #emFeedback.commands.stateComplete := NOT (NOT #tempScInProduction AND NOT #tempScNoProduction);
   #emFeedback.status.stateComplete := #emFeedback.commands.stateComplete;
   "Unit1.Em0.ControlNodes".em.status.stateComplete := #emFeedback.commands.stateComplete;
END_REGION

REGION Network 71: stateCommand Hold Summary
   RUNG wire#powerrail
      Contact( #statUnitStatus.mode.production )
      Contact( #statUnitStatus.state.execute )
      Contact( "Unit1.Em0.Alarms".materialFault[0] )
      Coil( #emFeedback.commands.hold )
   END_RUNG
   // the same network as SCL:
   #emFeedback.commands.hold := #statUnitStatus.mode.production AND #statUnitStatus.state.execute AND "Unit1.Em0.Alarms".materialFault[0];
END_REGION

REGION Network 72: *************** Alarms **********************************
END_REGION

REGION Network 73: Manage Alarms
   // Derive commands from the ProDiag supervision. The ProDiag supervisions contain categories which define the reaction of these supervisions (e.g. abort, stop, hold). These are handed over as commands to the unit level.
   // Alternatively, if no ProDiag should be used, you can use the LAF_ManageBitAlarms to realize bit alarm handling. This block can be found in LAF in folder 70_AlarmHandling.
